    DwellTimer(IN:=TRUE, PT:= T#10S);
	IF (DwellTimer.Q) THEN
		ErrorReturnState := ePistonInsertStaState.eRetractPalletHoldDownAndBarrel;		
		ResetDwellTimer();
		ResetStateTimer();
		NextState := ePistonInsertStaState.eError;		
	END_IF 
  

ePistonInsertStaState.eDepart:
	StateTimer(IN:=TRUE, PT:= T#20MS);
	IF (StateTimer.Q) THEN
		Stations.fbRoutePlanner.M_NotifyVehStaCmpl(StationIndex:= MM_CONST.PISTON_STA, VehicleID := VUT);
		xTrigger := FALSE;	
		StateTimer(IN:=FALSE);
		IF (NOT Stations.fbCycleControl.StopRequested) THEN			
			NextState := ePistonInsertStaState.eInit;
		ELSE 
			NextState := ePistonInsertStaState.eStopActive;
		END_IF
	END_IF

ePistonInsertStaState.eStopActive:
IF (NOT Stations.fbCycleControl.StopRequested) THEN			
	NextState := ePistonInsertStaState.eInit;
END_IF	
Status.PistonStatusMsg:= 'Piston Sta Cycle Stop, Hit Start'; 
	
ePistonInsertStaState.eError:
	Status.StationStauts[MM_CONST.PISTON_STA_HMI_STATE] := OverallStationStatus.eError;
	IF (GVL_IO.MC_XStartPB) THEN
		NextState := ErrorReturnState;
		ErrorReturnState := ePistonInsertStaState.eUnknown;
	END_IF

END_CASE

IF (State <> NextState) THEN
	bFirst := TRUE;
	StateTimer(IN:=FALSE);
ELSE
	bFirst := FALSE;
END_IF

State := NextState;
AssignStationStatusForHMI();

ACTION Act_EngagePalletHoldDown:
GVL_IO.PI_YPalletHoldDownExtend:= TRUE;
GVL_IO.PI_YPalletHoldDownRetract := FALSE;
END_ACTION

ACTION Act_ExtendBarrelBackup:
GVL_IO.PI_YBarrelBackupExtend := TRUE;
GVL_IO.PI_YBarrelBackupRetract := FALSE;
END_ACTION

ACTION Act_FreePalletHoldDown:
GVL_IO.PI_YPalletHoldDownExtend:= FALSE;
GVL_IO.PI_YPalletHoldDownRetract := TRUE;
END_ACTION

ACTION Act_RetractBarrelBackup:
GVL_IO.PI_YBarrelBackupExtend := FALSE;
GVL_IO.PI_YBarrelBackupRetract := TRUE;
END_ACTION

ACTION Act_SendEscapementToBowl:
GVL_IO.PI_YEscapementToBowl := TRUE;
GVL_IO.PI_YEscapementToWork := FALSE;
END_ACTION

ACTION Act_SendEscapementtoWork:
GVL_IO.PI_YEscapementToBowl := FALSE;
GVL_IO.PI_YEscapementToWork := TRUE;
END_ACTION

METHOD PUBLIC AssignStationStatusForHMI : BOOL
VAR_INPUT
END_VAR
Status.StationsState[MM_CONST.PISTON_STA_HMI_STATE] := State;
IF (NOT LotsData.Lot.PistonInsertEnabled AND NOT (State = ePistonInsertStaState.eUnknown) AND NOT (State = ePistonInsertStaState.eError)) THEN
	Status.StationStauts[MM_CONST.PISTON_STA_HMI_STATE] := OverallStationStatus.eDisabled;
ELSE 
	CASE State OF 
	ePistonInsertStaState.eUnknown,ePistonInsertStaState.eError: 
		Status.StationStauts[MM_CONST.PISTON_STA_HMI_STATE] := OverallStationStatus.eError;
	 
    
    ePistonInsertStaState.eSMCMtrReset,ePistonInsertStaState.eSMCMtrCheckEnabled,ePistonInsertStaState.eSMCMtrSendHome,
    ePistonInsertStaState.eSMCMtrHomed,ePistonInsertStaState.eInit, ePistonInsertStaState.eHoming,
	ePistonInsertStaState.eMoveEscapemttoBowl,
	ePistonInsertStaState.eEscapmentAtBowl,
	ePistonInsertStaState.eMoveEscapmentToWork,
	ePistonInsertStaState.eEscapementAtWork:
    	Status.StationStauts[MM_CONST.PISTON_STA_HMI_STATE] := OverallStationStatus.eHoming;	
	
	ePistonInsertStaState.eWaitForPartAtBowl:
		Status.StationStauts[MM_CONST.PISTON_STA_HMI_STATE] := OverallStationStatus.eWarning;
	
	ePistonInsertStaState.eReady:
		Status.StationStauts[MM_CONST.PISTON_STA_HMI_STATE] := OverallStationStatus.eWaitingForParts;
	
	ePistonInsertStaState.ePalletHoldDownEngaged,
	ePistonInsertStaState.eFirePistonUp,
	ePistonInsertStaState.eSendBarrelBackupEngage,
	ePistonInsertStaState.eWaitForPistonStartMovUp,
	ePistonInsertStaState.eWaitForBarrelBackupEngaged,
	ePistonInsertStaState.eWaitForPistonMovDoneUp,
	ePistonInsertStaState.eFirePistonDown,
	ePistonInsertStaState.eRetractPalletHoldDownAndBackup,
	ePistonInsertStaState.eWaitForPistonStartMovDwn,
	ePistonInsertStaState.eRetractPalletHoldDownAndBarrel,
	ePistonInsertStaState.eWaitForPalletHoldDownAndBackupRetracted,
	ePistonInsertStaState.eWaitForPistonMovDoneDown :
		Status.StationStauts[MM_CONST.PISTON_STA_HMI_STATE] := OverallStationStatus.eWaitingForParts; 
	
    ePistonInsertStaState.eStopActive:
	    Status.StationStauts[MM_CONST.PISTON_STA_HMI_STATE] := OverallStationStatus.eCycleStop;
	 
	ELSE ;
	
	END_CASE
END_IF
END_METHOD

METHOD PUBLIC ClearVehicleTrigger : BOOL
VAR_INPUT
END_VAR
xTrigger := FALSE;
END_METHOD

METHOD PUBLIC IsBarrelBackupExtended : BOOL
VAR_INPUT
END_VAR
IsBarrelBackUpExtended := TRUE;  // IMBAD 2 Has No Barrel Backup
(*
IsBarrelBackUpExtended := GVL_IO.PI_XBarrelHoldDownExtended AND NOT GVL_IO.PI_XBarrelHoldDownHome;
IF (NOT IsBarrelBackUpExtended) THEN
	Status.PistonStatusMsg := 'Piston: Check Barrel Backup Sensors';
END_IF
*)
END_METHOD

METHOD PUBLIC IsBarrelBackUpRetracted : BOOL
VAR_INPUT
END_VAR
IsBarrelBackUpRetracted := TRUE;  // IMBAD 2 has no Barrel Backup
(* 
IsBarrelBackUpRetracted := NOT GVL_IO.PI_XBarrelHoldDownExtended AND GVL_IO.PI_XBarrelHoldDownHome;
IF (NOT IsBarrelBackUpRetracted) THEN
	Status.PistonStatusMsg := 'Piston: Check Barrel Backup Sensors';
END_IF
*)
END_METHOD

METHOD PUBLIC IsEscapementAtBowl : BOOL
VAR_INPUT
END_VAR
IsEscapementAtBowl := (GVL_IO.PI_XEscapementAtBowl);// AND NOT GVL_IO.PI_XEscapementAtInsertLoc);
IF (NOT IsEscapementAtBowl) THEN
	Status.PistonStatusMsg := 'Piston: Check Escapment Sensors';
END_IF
END_METHOD

METHOD PUBLIC IsEscapementAtWork : BOOL
VAR_INPUT
END_VAR
IsEscapementAtWork := ((*NOT GVL_IO.PI_XEscapementAtBowl AND *)GVL_IO.PI_XEscapementAtInsertLoc);
IF (NOT IsEscapementAtWork) THEN
	Status.PistonStatusMsg := 'Piston: Check Escapment Sensors';
END_IF
END_METHOD

METHOD PUBLIC IsFaulted : BOOL
VAR_INPUT
END_VAR
IsFaulted := (State = ePistonInsertStaState.eUnknown OR State = ePistonInsertStaState.eError);
END_METHOD

METHOD PUBLIC IsPalletHoldDownEngaged : BOOL
VAR_INPUT
END_VAR
IsPalletHoldDownEngaged := (NOT GVL_IO.PI_XPalletHoldDownHome (*AND GVL_IO.PI_XPalletHoldDownExtended*));
IF (NOT IsPalletHoldDownEngaged) THEN
	Status.PistonStatusMsg := 'Piston: Check Pallet Hold Down'; 
END_IF
END_METHOD

METHOD PUBLIC IsPalletHoldDownFree : BOOL
VAR_INPUT
END_VAR
IsPalletHoldDownFree := (GVL_IO.PI_XPalletHoldDownHome AND NOT GVL_IO.PI_XPalletHoldDownExtended);
IF (NOT IsPalletHoldDownFree) THEN
	Status.PistonStatusMsg := 'Piston: Check Pallet Hold Down'; 
END_IF
END_METHOD

METHOD PUBLIC LEY_MasterReset : BOOL
VAR_INPUT
END_VAR
GVL_IO.PI_YMtrReset := TRUE;
GVL_IO.PI_YMtrSetEnable:= TRUE;
GVL_IO.PI_YMtrDriveStepTrigger := FALSE;
GVL_IO.PI_YMtrHoldMove := FALSE;
GVL_IO.PI_YMtrGoHome := FALSE;
GVL_IO.PI_YMtrJogNeg := FALSE;
GVL_IO.PI_YMtrJogPos := FALSE;
GVL_IO.PI_YMtrSwitchJogInch := FALSE;
GVL_IO.PI_YMtrStepSelectIN0:= FALSE;
GVL_IO.PI_YMtrStepSelectIN1:= FALSE;
GVL_IO.PI_YMtrStepSelectIN2:= FALSE;
GVL_IO.PI_YMtrStepSelectIN3:= FALSE;
GVL_IO.PI_YMtrStepSelectIN4:= FALSE;
GVL_IO.PI_YMtrStepSelectIN5:= FALSE;
END_METHOD

PROPERTY PUBLIC Ready : BOOL
GET
IF (LotsData.Lot.PistonInsertEnabled) THEN
	Ready := (State = ePistonInsertStaState.eReady);
ELSE
    Ready := (State = ePistonInsertStaState.eDisabledReady);
END_IF
END_GET
END_PROPERTY

ACTION ResetDwellTimer:
DwellTimer(IN:=FALSE);
END_ACTION

METHOD PUBLIC ResetState : BOOL
VAR_INPUT
END_VAR
	State := ePistonInsertStaState.eUnknown;
	NextState := ePistonInsertStaState.eUnknown;
END_METHOD

ACTION ResetStateTimer:
StateTimer(IN:=FALSE);
END_ACTION

PROPERTY PUBLIC Trigger : BOOL
SET
xTrigger := Trigger;
END_SET
END_PROPERTY

METHOD PUBLIC UpdatePartData : BOOL
VAR_INPUT
END_VAR
PartsData.Status[VUT].OverallStatus := ePartStatus.ePistonInserted;
PartsData.Status[VUT].PistonStroke := GVL_IO.PI_XMtrCurrPos;
PartsData.Status[VUT].PistonPass := TRUE;
PartsData.Status[VUT].PistonInsertTime := SYSTEMTIME_TO_STRING(Logging.fbCurrTime.systemTime);
END_METHOD

PROPERTY PUBLIC VehicleUnderTest : BYTE
GET
VehicleUnderTest := VUT;
END_GET
SET
VUT := VehicleUnderTest;
END_SET
END_PROPERTY

END_FUNCTION_BLOCK

// ---- POUs/IB_StopRobotClearStation.TcPOU
FUNCTION_BLOCK PUBLIC IB_StopRobotClearStation
VAR_INPUT
END_VAR
VAR_OUTPUT
END_VAR
VAR
	xTrigger :BOOL := FALSE; // triggers processing
	State : eIB_StopRobotClearStaState := eIB_StopRobotClearStaState.eUnknown;
	NextState : eIB_StopRobotClearStaState := eIB_StopRobotClearStaState.eUnknown;
	bFirst : BOOL := TRUE;
	VUT : BYTE; //VehicleID Under Station
	DwellTimer : TON;
END_VAR

CASE State OF
eIB_StopRobotClearStaState.eUnknown:
	NextState := eIB_StopRobotClearStaState.eReady;
	
eIB_StopRobotClearStaState.eInit:

eIB_StopRobotClearStaState.eHoming:

eIB_StopRobotClearStaState.eReady:
	IF (xTrigger) THEN
		NextState := eIB_StopRobotClearStaState.eProcessing;		
		DwellTimer(IN:=FALSE);
	END_IF

eIB_StopRobotClearStaState.eDwell:	

eIB_StopRobotClearStaState.eProcessing:
	IF(Stations.fbLoad1Sta.HoldVehicle_IBStop = FALSE) THEN
		NextState := eIB_StopRobotClearStaState.eDepart;
	END_IF

eIB_StopRobotClearStaState.eDepart:
		Stations.fbRoutePlanner.M_NotifyVehStaCmpl(StationIndex:= MM_CONST.IB_STOP_ROBOT_CLEAR_STA, VehicleID := VUT);
		xTrigger := FALSE;
		IF (Stations.fbCycleControl.StopRequested) THEN
			NextState := eIB_StopRobotClearStaState.eStopActive;
		ELSE
			NextState := eIB_StopRobotClearStaState.eReady;		
		END_IF
		
eIB_StopRobotClearStaState.eStopActive:
	IF (NOT Stations.fbCycleControl.StopRequested) THEN
		NextState := eIB_StopRobotClearStaState.eReady;	
	END_IF
		
eIB_StopRobotClearStaState.eError:
END_CASE

IF (State <> NextState) THEN
	bFirst := TRUE;
ELSE
	bFirst := FALSE;
END_IF

State := NextState;
//Status.StationsState[MM_CONST.IB_STOP_ROBOT_CLEAR_STA_HMI_STATE] := State;
//AssignStationStatusForHMI();

METHOD PUBLIC ClearVehicleTrigger : BOOL
VAR_INPUT
END_VAR
xTrigger := FALSE;
State  := eIB_StopRobotClearStaState.eUnknown;
NextState  := eIB_StopRobotClearStaState.eUnknown;
bFirst  := TRUE;
END_METHOD

PROPERTY PUBLIC Trigger : BOOL
SET
xTrigger := Trigger;
END_SET
END_PROPERTY

PROPERTY PUBLIC VehicleUnderTest : BYTE
GET
VehicleUnderTest := VUT;
END_GET
SET
VUT := VehicleUnderTest;
END_SET
END_PROPERTY

END_FUNCTION_BLOCK

// ---- POUs/CapInsertStation.TcPOU
FUNCTION_BLOCK PUBLIC CapInsertStation
VAR_INPUT
END_VAR
VAR_OUTPUT
END_VAR
VAR
	xTrigger :BOOL := FALSE; // triggers processing
	State : eCapInsertStaState := eCapInsertStaState.eUnknown;
	NextState : eCapInsertStaState := eCapInsertStaState.eUnknown;
	ErrorReturnState :  eCapInsertStaState := eCapInsertStaState.eUnknown;
	bFirst : BOOL := TRUE;
	VUT : BYTE; //VehicleID Under Station
	DwellTimer : TON;		
	StateTimer : TON;
	PartPresentTimer : TON;
	CapInstallRetries : BYTE :=0;
	CapPickUpRetries : BYTE := 0;
	CapTorqueTime : TIME := T#250MS;
END_VAR

/// Cap station can be either Disabled or Enabled
// If Disabled, then we need to be in a state such that it is disabled but will not cause any obstacles. 
// Either in Disabled - Ready or Enabled- Ready, provide a way to account for Station enable change

IF (GVL_IO.MachineEStopped) THEN 
	State := eCapInsertStaState.eUnknown;
	NextState := eCapInsertStaState.eUnknown;	
END_IF

CASE State OF

eCapInsertStaState.eUnknown:
	   IF (GVL_IO.MC_XStartPB AND GVL_IO.MC_XAirPressureOK AND GVL_IO.MC_NotEStopped) THEN // wait for start button when powered up or PLC program restarted
		 ResetDwellTimer();	
         NextState := eCapInsertStaState.eHoming;	              
	   END_IF
	ACT_RetractSlide();
	ACT_RetractPalletHoldDown();
	Status.CapStatusMsg:= 'CapSta Unknown,Check Air/E-STOP THEN Hit Start';

eCapInsertStaState.eHoming:
    Status.StationStauts[MM_CONST.CAP_STA_HMI_STATE] := OverallStationStatus.eHoming;
	Status.CapStatusMsg:= 'Cap Station Homing';
	
	ACT_RetractSlide();
	ACT_RetractPalletHoldDown();
	DwellTimer(IN:=TRUE, PT:= T#10S);	
	IF (IsPalletHoldDownRetracted() AND IsSlideRetracted()) THEN
		ResetDwellTimer();	
		IF (NOT LotsData.Lot.CapInsertEnabled) THEN
			NextState :=  eCapInsertStaState.eDisabledReady;			
        ELSE 
            NextState :=  eCapInsertStaState.eWaitForVehicleTrigger;
		END_IF
	END_IF
    IF (DwellTimer.Q) THEN
		ResetDwellTimer();
		NextState := eCapInsertStaState.eError;
		ErrorReturnState := eCapInsertStaState.eHoming;		
	END_IF
	
	

eCapInsertStaState.eDisabledReady:
	ACT_RetractSlide();
	ACT_RetractPalletHoldDown();
	IF (LotsData.Lot.CapInsertEnabled) THEN 
		NextState := eCapInsertStaState.eUnknown; // force the operator to hit the start button if station is enabled.
	END_IF
	IF (xTrigger) THEN // vehicles that have been previously commanded to come here before station was disabled 
		NextState := eCapInsertStaState.eDepart;
	END_IF
	Status.StationStauts[MM_CONST.CAP_STA_HMI_STATE] := OverallStationStatus.eDisabled;
	Status.CapStatusMsg:= 'Cap Station Disabled and Clear for pallets to move';
	
	
eCapInsertStaState.eWaitForVehicleTrigger:
  
	IF (xTrigger) THEN //XTrigger is signaled when part arrives under the station
		NextState := eCapInsertStaState.ePalletHoldDownGoingDown;	
	    PartsData.Status[VUT].OverallStatus := ePartStatus.eReject; 		
		ResetDwellTimer();
	END_IF
	
	Status.StationStauts[MM_CONST.CAP_STA_HMI_STATE] := OverallStationStatus.eWaitingForParts;
	Status.CapStatusMsg:= 'Cap Station Waiting For Parts';

eCapInsertStaState.ePalletHoldDownGoingDown:
	ACT_EngagePalletHoldDown();
	IF (IsPalletHoldDownExtended()) THEN
		   NextState := eCapInsertStaState.ePalletHoldDownExtended;		 
           ResetDwellTimer();  
	   END_IF
	DwellTimer(IN:=TRUE, PT:= T#10S); // give a message out every 10 seconds
	IF (DwellTimer.Q) THEN
		ResetDwellTimer();
		NextState := eCapInsertStaState.eError;
		ErrorReturnState := eCapInsertStaState.ePalletHoldDownGoingDown;			
	END_IF
	
	Status.StationStauts[MM_CONST.CAP_STA_HMI_STATE] := OverallStationStatus.eRunning;
	Status.CapStatusMsg:= 'Cap Cycle In Progress';
	
eCapInsertStaState.ePalletHoldDownExtended:
   DwellTimer(IN:=TRUE, PT:= T#250MS);
   IF (DwellTimer.Q) THEN 
	   ResetDwellTimer();
       NextState := eCapInsertStaState.eCapSlideGoingDown;
   END_IF

eCapInsertStaState.eCapSlideGoingDown:
   ACT_ExtendSlide();
   IF (NOT IsSlideRetracted()) THEN 
	   NextState := eCapInsertStaState.eCapSlideExtended;
	   ResetDwellTimer();
   END_IF
   DwellTimer(IN:=TRUE, PT:= T#5S); // give a message out every 10 seconds
	IF (DwellTimer.Q) THEN
		ResetDwellTimer();
		Act_RetractSlide();  // Not wanting to spin the cap station if case of time out
		NextState := eCapInsertStaState.eError;
		ErrorReturnState := eCapInsertStaState.eCapSlideGoingDown;			
	END_IF

eCapInsertStaState.eCapSlideExtended:
   DwellTimer(IN:=TRUE, PT:= CapTorqueTime);
   IF (DwellTimer.Q OR IsSlideExtended()) THEN 
	   ResetDwellTimer();
	   UpdatePartData();	   
       NextState := eCapInsertStaState.eCapSlideGoingUp;
   END_IF

 eCapInsertStaState.eCapSlideGoingUp:
   ACT_RetractSlide();
   ResetDwellTimer();
   NextState := eCapInsertStaState.eCapSlideUp;
   
eCapInsertStaState.eCapSlideUp:
    IF (IsSlideRetracted()) THEN
	   ResetDwellTimer();
	   NextState := eCapInsertStaState.ePalletHoldDownGoingUp;
   END_IF
   
    DwellTimer(IN:=TRUE, PT:= T#10S); 
	IF (DwellTimer.Q) THEN
		ResetDwellTimer();
		NextState := eCapInsertStaState.eError;
		ErrorReturnState := eCapInsertStaState.eCapSlideGoingUp;			
	END_IF
   
eCapInsertStaState.ePalletHoldDownGoingUp:
	ACT_RetractPalletHoldDown();
	ResetDwellTimer();
	NextState := eCapInsertStaState.ePalletHoldDownUp;

eCapInsertStaState.ePalletHoldDownUp:
  
   IF (IsPalletHoldDownRetracted()) THEN
	   ResetDwellTimer();
	   NextState := eCapInsertStaState.eDepart;
   END_IF 
    DwellTimer(IN:=TRUE, PT:= T#10S); // give a message out every 10 seconds
	IF (DwellTimer.Q) THEN
		ResetDwellTimer();
		NextState := eCapInsertStaState.eError;
		ErrorReturnState := eCapInsertStaState.ePalletHoldDownGoingUp;			
	END_IF


eCapInsertStaState.eDepart:
	Stations.fbRoutePlanner.M_NotifyVehStaCmpl(StationIndex:= MM_CONST.CAP_STA, VehicleID := VUT);
	xTrigger := FALSE; // Now that we have sent a vehicle out, we should not work on it anymore 
    IF (Stations.fbCycleControl.StopRequested) THEN		
		NextState := eCapInsertStaState.eStopActive;
	ELSE
		NextState := eCapInsertStaState.eHoming;
	END_IF

eCapInsertStaState.eStopActive:
IF (NOT Stations.fbCycleControl.StopRequested) THEN		
		NextState := eCapInsertStaState.eHoming;
END_IF	
    Status.StationStauts[MM_CONST.CAP_STA_HMI_STATE] := OverallStationStatus.eCycleStop;	
    Status.CapStatusMsg:= 'Cap Stop Active, Press Start to Run';
	
eCapInsertStaState.eError:
	Status.StationStauts[MM_CONST.CAP_STA_HMI_STATE] := OverallStationStatus.eError;
	IF (GVL_IO.MC_XStartPB) THEN
		NextState := ErrorReturnState;
		ErrorReturnState := eCapInsertStaState.eUnknown;
	END_IF
	
END_CASE

IF (State <> NextState) THEN
	bFirst := TRUE;
	StateTimer(IN:=FALSE);
ELSE
	bFirst := FALSE;
END_IF

State := NextState;

ACTION ACT_EngagePalletHoldDown:
GVL_IO.CP_YPalletHoldDownExtend := TRUE;
GVL_IO.CP_YPalletHoldDownRetract := FALSE;
END_ACTION

ACTION ACT_ExtendSlide:
GVL_IO.CP_YCapSlideExtend := TRUE;
GVL_IO.CP_YCapSlideRetract := FALSE;
END_ACTION

ACTION ACT_RetractPalletHoldDown:
GVL_IO.CP_YPalletHoldDownExtend := FALSE;
GVL_IO.CP_YPalletHoldDownRetract := TRUE;
END_ACTION

ACTION ACT_RetractSlide:
GVL_IO.CP_YCapSlideExtend := FALSE;
GVL_IO.CP_YCapSlideRetract := TRUE;
END_ACTION

METHOD PUBLIC ClearVehicleTrigger : BOOL
VAR_INPUT
END_VAR
xTrigger := FALSE;
END_METHOD

METHOD PUBLIC IsFaulted : BOOL
VAR_INPUT
END_VAR
IF (LotsData.Lot.CapInsertEnabled) THEN 
	IsFaulted := (State = eCapInsertStaState.eUnknown OR State = eCapInsertStaState.eError);
ELSE 
	IsFaulted := FALSE;
END_IF
END_METHOD

METHOD PUBLIC IsPalletHoldDownExtended : BOOL
VAR_INPUT
END_VAR
IsPalletHoldDownExtended := (GVL_IO.CP_XPalletHoldDownExtended AND NOT GVL_IO.CP_XPalletHoldDownHome);
IF (NOT IsPalletHoldDownExtended) THEN 
	Status.CapStatusMsg := 'Cap Station: Check Pallet HoldDown Sensors'; 
END_IF
END_METHOD

METHOD PUBLIC IsPalletHoldDownRetracted : BOOL
VAR_INPUT
END_VAR
IsPalletHoldDownRetracted := (NOT GVL_IO.CP_XPalletHoldDownExtended AND GVL_IO.CP_XPalletHoldDownHome);
IF (NOT IsPalletHoldDownRetracted) THEN 
	Status.CapStatusMsg := 'Cap Station: Check Pallet HoldDown Sensors'; 
END_IF
END_METHOD

METHOD IsSlideExtended : BOOL
VAR_INPUT
END_VAR
IsSlideExtended := (GVL_IO.CP_XCapSlideExtended AND NOT GVL_IO.CP_XCapSlideRetracted);
IF (NOT IsSlideExtended) THEN 
	Status.CapStatusMsg := 'Cap Station: Check Slide Sensors'; 
END_IF
END_METHOD

METHOD PUBLIC IsSlideRetracted : BOOL
VAR_INPUT
END_VAR
//IsSlideRetracted := TRUE; //turnkey slide removed

IsSlideRetracted := (NOT GVL_IO.CP_XCapSlideExtended AND GVL_IO.CP_XCapSlideRetracted);
IF (NOT IsSlideRetracted) THEN 
	Status.CapStatusMsg := 'Cap Station: Check Slide Sensors'; 
END_IF
END_METHOD

PROPERTY PUBLIC Ready : BOOL
GET
IF (LotsData.Lot.CapInsertEnabled) THEN
 Ready := (State = eCapInsertStaState.eWaitForVehicleTrigger);
ELSE
	Ready := (State = eCapInsertStaState.eDisabledReady);	//we removed the physical cap station on 10/17 
END_IF
END_GET
END_PROPERTY

ACTION ResetDwellTimer:
DwellTimer(IN:=FALSE);
END_ACTION

METHOD PUBLIC ResetState : BOOL
VAR_INPUT
END_VAR
	State := eCapInsertStaState.eUnknown;
	NextState := eCapInsertStaState.eUnknown;
	ErrorReturnState := eCapInsertStaState.eUnknown;
END_METHOD

PROPERTY PUBLIC Trigger : BOOL
SET
xTrigger := Trigger;
END_SET
END_PROPERTY

METHOD PUBLIC UpdatePartData : BOOL
VAR_INPUT
END_VAR
IF ( NOT IsSlideExtended()) THEN
	PartsData.Status[VUT].OverallStatus := ePartStatus.eCapInserted;
	PartsData.Status[VUT].CapPass := TRUE;
	PartsData.Status[VUT].CapInsertTime := SYSTEMTIME_TO_STRING(Logging.fbCurrTime.systemTime);	
ELSE // there is no cap
	PartsData.Status[VUT].OverallStatus := ePartStatus.eReject;
	PartsData.Status[VUT].CapPass := FALSE;
	PartsData.Status[VUT].CapInsertTime := SYSTEMTIME_TO_STRING(Logging.fbCurrTime.systemTime);
END_IF
END_METHOD

PROPERTY PUBLIC VehicleUnderTest : BYTE
GET
VehicleUnderTest := VUT;
END_GET
SET
VUT := VehicleUnderTest;
END_SET
END_PROPERTY

END_FUNCTION_BLOCK

// ---- POUs/GoodUnloadStation.TcPOU
FUNCTION_BLOCK PUBLIC GoodUnloadStation
VAR_INPUT
END_VAR
VAR_OUTPUT
END_VAR
VAR
	xTrigger :BOOL := FALSE; // triggers processing
	State : eGoodULStaState := eGoodULStaState.eUnknown;
	NextState : eGoodULStaState := eGoodULStaState.eUnknown;	
	ErrorReturnState : eGoodULStaState := eGoodULStaState.eUnknown;	
	bFirst : BOOL := TRUE;
	VUT : BYTE; //VehicleID Under Station
	DwellTimer : TON;
	StateTimer : TON;
	eDwell: INT;
	eDepart: INT;
	CurrPPLoc : BYTE;
	GripperOpenTimer :TIME := T#200MS;
	//StopAfter
	DropLocation : BYTE;
	GoodFullCount : UINT := 0;
	PremiumFullCount : UINT := 0;
	
END_VAR

IF (GVL_IO.MachineEStopped) THEN 
	State := eGoodULStaState.eUnknown;
	NextState := eGoodULStaState.eUnknown;	
	Status.GoodULStatusMsg:= 'Unload: Unknown State, Check E-STOP, Check Air, Hit Start';
END_IF

GetPPLocation(Location=>CurrPPLoc); // Get where PP Location is from the Bits. 

IF (NOT LotsData.Lot.AutoBaggerEnabled) THEN
	Config.PremiumCount1 := 0;
	Config.PremiumCount2 := 0;
	Config.GoodCount1 := 0;
	Config.GoodCount2 := 0;
	GoodFullCount := 0;
    PremiumFullCount := 0;
END_IF


CASE State OF
	
eGoodULStaState.eUnknown:
	IF (GVL_IO.MC_XStartPB AND GVL_IO.MC_XAirPressureOK AND GVL_IO.MC_NotEStopped) THEN // wait for start button when powered up or PLC program restarted
			NextState := eGoodULStaState.eInit;	   
	END_IF

eGoodULStaState.eInit:
    Act_OpenGrippers();
	Act_FreePalletHold();
	Act_FreePalletRelease();
    Act_MoveRotatorCenter();
	Act_ResetPPIO();	
	
	StateTimer(IN:=TRUE,PT:= T#100MS);
	IF (StateTimer.Q) THEN
		NextState := eGoodULStaState.eHoming;
		ResetStateTimer();
	END_IF	

eGoodULStaState.eHoming:
  
	IF (IsGripperOpen() AND IsPalletReleaseFree() AND IsRotatorCenter() AND IsPalletHoldDownFree()) THEN
	  NextState := eGoodULStaState.eHPReset;
	  ResetDwellTimer();
 	END_IF	
	
   DwellTimer(IN:=TRUE, PT:= T#10S);
   IF (DwellTimer.Q) THEN
		ErrorReturnState := eGoodULStaState.eInit;		
		ResetDwellTimer();
		ResetStateTimer();
        NextState := eGoodULStaState.eError;		
	END_IF
	

eGoodULStaState.eHPReset:
	IF (GVL_IO.UL_XPP_Alarm) THEN
		DwellTimer(IN:= TRUE, PT := T#2S);	
	END_IF
	IF (DwellTimer.Q) THEN
		ResetDwellTimer();
		GVL_IO.UL_YPP_ResetAlarm := NOT GVL_IO.UL_YPP_ResetAlarm; // toggle the reset request every four seconds 
	END_IF
	IF (NOT GVL_IO.UL_XPP_Alarm) THEN
		GVL_IO.UL_YPP_Enable:= TRUE;
		GVL_IO.UL_YPP_ResetAlarm := FALSE;
		ResetDwellTimer();
		NextState := eGoodULStaState.eHPCheckEnabled;	
	END_IF
	// Time out condition... hang here until Pick Place Alarm is reset... 
	DwellTimer(IN:=TRUE, PT:= T#10S);
   IF (DwellTimer.Q) THEN
		ErrorReturnState := eGoodULStaState.eHPReset;		
		ResetDwellTimer();
		ResetStateTimer();
		Status.GoodULStatusMsg:= 'Pick&Place unable to Reset';
        NextState := eGoodULStaState.eError;		
	END_IF

eGoodULStaState.eHPCheckEnabled:
	IF (GVL_IO.UL_XPP_DriveEnabled AND NOT GVL_IO.UL_XPP_Alarm) THEN
		ResetDwellTimer();
        IF (GVL_IO.UL_XPP_ReferenceOK) THEN
			NextState := eGoodULStaState.eHPHomed;			
			GVL_IO.UL_YPP_StartHoming := FALSE;
		ELSE			
			NextState := eGoodULStaState.eHPSendHome;
		END_IF
	END_IF
	
	// Time out condition... hang here until Pick Place Alarm is reset... 
   DwellTimer(IN:=TRUE, PT:= T#10S);
   IF (DwellTimer.Q) THEN
		ErrorReturnState := eGoodULStaState.eHPReset;		
		ResetDwellTimer();
		ResetStateTimer();
		Status.GoodULStatusMsg:= 'Pick&Place unable to Enable';
        NextState := eGoodULStaState.eError;		
	END_IF

eGoodULStaState.eHPSendHome:
	GVL_IO.UL_YPP_Stop := FALSE;
	IF (NOT GVL_IO.UL_XPP_StopActive AND GVL_IO.UL_XPP_ReadyToStart AND GVL_IO.UL_XPP_DriveEnabled AND NOT GVL_IO.UL_XPP_Alarm) THEN
		GVL_IO.UL_YPP_StartHoming := TRUE;
	END_IF
	
   IF (GVL_IO.UL_XPP_ReferenceOK) THEN
	   NextState := eGoodULStaState.eHPHomed;
	   ResetDwellTimer();
   END_IF
   
   DwellTimer(IN:=TRUE, PT:= T#2M);
   IF (DwellTimer.Q) THEN
		ErrorReturnState := eGoodULStaState.eInit;		
		ResetDwellTimer();
		ResetStateTimer();
		GVL_IO.UL_YPP_StartHoming := FALSE;
		Status.GoodULStatusMsg:= 'Pick&Place unable to Home';
        NextState := eGoodULStaState.eError;		
	END_IF
 

eGoodULStaState.eHPHomed:
	GVL_IO.UL_YPP_Stop := FALSE;
	GVL_IO.UL_YPP_Enable := TRUE;
	GVL_IO.UL_YPP_StartHoming := FALSE;
	IF (GVL_IO.UL_XPP_ReadyToStart) THEN
		NextState := eGoodULStaState.eHPSendToInitLoc;
		ResetDwellTimer();
		ResetStateTimer();
	END_IF
	
    DwellTimer(IN:=TRUE, PT:= T#2M);
   IF (DwellTimer.Q) THEN
		ErrorReturnState := eGoodULStaState.eHPReset;		
		ResetDwellTimer();
		ResetStateTimer();
		GVL_IO.UL_YPP_StartHoming := FALSE;
		Status.GoodULStatusMsg:= 'Pick&Place unable to Ready To Start';
        NextState := eGoodULStaState.eError;		
	END_IF

eGoodULStaState.eHPSendToInitLoc:
   // we have to set Seq 1 as InitLoc ( Up at Pick Location). Also, Input bits will corresponding to the sequence 
   SetPPSequence(SequenceNumb := 1);
   DwellTimer(IN:= TRUE, PT:= T#30MS);
   IF (DwellTimer.Q) THEN
	   GVL_IO.UL_YPP_StartSeq := TRUE;
	   ResetDwellTimer();
   END_IF
   StateTimer(IN:= GVL_IO.UL_YPP_StartSeq, PT:= T#30MS);
   IF (StateTimer.Q) THEN
	   NextState := eGoodULStaState.eHPAtInitLoc;
	   ResetStateTimer();
	   ResetDwellTimer();
   END_IF
 
eGoodULStaState.eHPAtInitLoc:
	IF (CurrPPLoc = 1) THEN
		NextState:= eGoodULStaState.eHPReady;
		GVL_IO.UL_YPP_StartSeq := FALSE;
		ResetDwellTimer();
		ResetStateTimer();
	END_IF
   DwellTimer(IN:=TRUE, PT:= T#10S);
   IF (DwellTimer.Q) THEN
		ErrorReturnState := eGoodULStaState.eHPSendToInitLoc;		
		ResetDwellTimer();
		ResetStateTimer();
		GVL_IO.UL_YPP_StartSeq := FALSE;
		Status.GoodULStatusMsg:= 'Pick&Place unable to Go To Init Loc';
        NextState := eGoodULStaState.eError;		
	END_IF

eGoodULStaState.eHPReady:
    Status.GoodULStatusMsg:= 'Unload Ready';
    Act_OpenGrippers();
	Act_FreePalletHold();
    Act_FreePalletRelease();
    Act_MoveRotatorCenter();	
	//PP fieldbus commands
	SetPPSequence(SequenceNumb := 1);
	Act_EnablePP();
	GVL_IO.UL_YPP_StartSeq := FALSE;
	
	 IF (IsGripperOpen() AND IsPalletReleaseFree() AND IsRotatorCenter() AND IsPalletHoldDownFree() AND GVL_IO.UL_XPP_ReadyToStart ) THEN
	  	 ResetDwellTimer();
         IF (LotsData.Lot.GoodUnloadEnabled) THEN
			 NextState:= eGoodULStaState.eWaitForVehicleTrigger;			 
		 ELSE 
			 NextState := eGoodULStaState.eDisabledReady;
		 END_IF    
    END_IF	
	
	DwellTimer(IN:=TRUE, PT:= T#10S);
   IF (DwellTimer.Q) THEN
		ErrorReturnState := eGoodULStaState.eHPReady;		
		ResetDwellTimer();
		ResetStateTimer();				
        NextState := eGoodULStaState.eError;		
	END_IF
	
	

eGoodULStaState.eDisabledReady:
	
	IF (LotsData.Lot.GoodUnloadEnabled) THEN
		NextState := eGoodULStaState.eUnknown;
	END_IF
	IF (xTrigger) THEN
		Stations.fbRoutePlanner.M_NotifyVehStaCmpl(StationIndex:= MM_CONST.GOOD_UNLOAD_STA, VehicleID := VUT);
		xTrigger := FALSE;
		NextState := eGoodULStaState.eDepartVehicle;
	END_IF

eGoodULStaState.eWaitForVehicleTrigger:

	IF (xTrigger) THEN //XTrigger is signaled when part arrives under the station
		DwellTimer(IN:=TRUE, PT:= T#100MS);
        IF (DwellTimer.Q) THEN 
			NextState := eGoodULStaState.eDetermineDropLocation;
			ResetDwellTimer();
        END_IF								
	END_IF
	
	IF (NOT LotsData.Lot.GoodUnloadEnabled) THEN
		NextState := eGoodULStaState.eDisabledReady;
	END_IF
	
	Status.GoodULStatusMsg:= 'Unload Ready: Waiting For Vehicle';
		 
eGoodULStaState.eDetermineDropLocation: //Determine drop locations.  Premiums can go in good if Premium is full.  

	IF (PartsData.Status[VUT].Premium) THEN
		IF (NOT LotsData.Lot.AutoBaggerEnabled) THEN
			DropLocation := 1;
			NextState := eGoodULStaState.eDwell;
		ELSIF ((Config.PremiumCount1 < LotsData.Lot.QuantityInBag) AND ((Config.PremiumCount2 < (LotsData.Lot.QuantityInBag-10)) OR (Config.PremiumCount2 = LotsData.Lot.QuantityInBag))) THEN
			DropLocation := 1;
			NextState := eGoodULStaState.eDwell;
			PremiumFullCount := 0;
		ELSIF (Config.PremiumCount2 < LotsData.Lot.QuantityInBag) THEN
			DropLocation := 2;
			NextState := eGoodULStaState.eDwell;
			PremiumFullCount := 0;
		ELSE
			PartsData.Status[VUT].Premium := FALSE;
			PartsData.Status[VUT].Good := TRUE;
			PremiumFullCount := PremiumFullCount + 1;
		END_IF
	END_IF
	
	IF (PartsData.Status[VUT].Good) THEN      /// remove this after Turnkey Debug
		IF (NOT LotsData.Lot.AutoBaggerEnabled) THEN
			DropLocation := 3;
			NextState := eGoodULStaState.eDwell;
		ELSIF ((Config.GoodCount1 < LotsData.Lot.QuantityInBag) AND ((Config.GoodCount2 < (LotsData.Lot.QuantityInBag-10)) OR (Config.GoodCount2 = LotsData.Lot.QuantityInBag))) THEN
			DropLocation := 3;
			NextState := eGoodULStaState.eDwell;
			GoodFullCount := 0;
		ELSIF (NOT (Config.GoodCount2 >= LotsData.Lot.QuantityInBag)) THEN
			DropLocation := 4;
			NextState := eGoodULStaState.eDwell;
			GoodFullCount := 0;
		ELSE
			PartsData.Status[VUT].Premium := FALSE;
			PartsData.Status[VUT].Good := FALSE;
			PartsData.Status[VUT].OverallStatus := ePartStatus.eReject;
			PartsData.Status[VUT].GoodUnload := FALSE;
			GoodFullCount := GoodFullCount + 1;
		END_IF	
	END_IF
    	
	IF (PartsData.Status[VUT].OverallStatus = ePartStatus.eReject) THEN
		NextState := eGoodULStaState.eAbandonCycle;
	END_IF	
	
	IF (GoodFullCount >= 5 OR PremiumFullCount >= 5) THEN
		Stations.fbCycleControl.StopRequested := TRUE;
		Status.AutoBaggerStatusMsg := 'AutoBagger: No drop location available.';
	END_IF
	

eGoodULStaState.eDwell:
    DwellTimer(IN:=GVL_IO.UL_XBarrelPresent, PT := T#50MS);  /// Need to add Part Data to get this status to find if part needs to be rejected
	IF (DwellTimer.Q) THEN		
        NextState := eGoodULStaState.eEngagePalletHoldDown;
		ResetDwellTimer();
		ResetStateTimer();
    END_IF
	StateTimer(IN:=TRUE, PT:= T#1S);
	IF (StateTimer.Q) THEN
		NextState := eGoodULStaState.eAbandonCycle;
		ResetStateTimer();
		ResetDwellTimer();
		//NextState := eGoodULStaState.eEngagePalletHoldDown;
	END_IF
	
 eGoodULStaState.eAbandonCycle:
 	Act_FreePalletHold();
	Act_FreePalletRelease();
	IF (IsPalletHoldDownFree() AND IsPalletReleaseFree()) THEN
		ResetDwellTimer();
        NextState := eGoodULStaState.eDepartVehicle;
		Stations.fbRoutePlanner.M_NotifyVehStaCmpl(StationIndex:= MM_CONST.GOOD_UNLOAD_STA, VehicleID := VUT);
		xTrigger:= FALSE;
	END_IF
	
   DwellTimer(IN:=TRUE, PT:= T#10S);
   IF (DwellTimer.Q) THEN
		ErrorReturnState := eGoodULStaState.eHPReset;		
		ResetDwellTimer();
		ResetStateTimer();		
        NextState := eGoodULStaState.eError;		
	END_IF
	
		
eGoodULStaState.eEngagePalletHoldDown:

	Act_EngagePalletHold();
	NextState := eGoodULStaState.ePalletHoldDownEngaged;;
	IF (IsPalletHoldDownEngaged()) THEN	 // speed up more, don't wait here
		NextState := eGoodULStaState.ePalletHoldDownEngaged;
        //NextState := eGoodULStaState.eAbandonCycle;		
	END_IF
	
eGoodULStaState.ePalletHoldDownEngaged:
	//NextState:= eGoodULStaState.ePalletReleaseExtend;
	NextState := eGoodULStaState.eHPMoveToPickFromTrack;
	ResetDwellTimer();
	ResetStateTimer();
	
eGoodULStaState.eHPMoveToPickFromTrack:
    SetPPSequence(SequenceNumb := 2); // Pick location    
	Act_MoveRotatorCenter(); // also move rotary while going down
   	DwellTimer(IN:= TRUE, PT:= T#20MS);
   	IF (DwellTimer.Q) THEN
	   GVL_IO.UL_YPP_StartSeq := TRUE;
	   ResetDwellTimer();
   END_IF
   StateTimer(IN:= GVL_IO.UL_YPP_StartSeq, PT:= T#20MS);
   IF (StateTimer.Q) THEN
	   NextState := eGoodULStaState.eHPAtPickFromTrack;
	   ResetDwellTimer();
	   ResetStateTimer();
   END_IF


eGoodULStaState.eHPAtPickFromTrack:
	IF (CurrPPLoc = 2 ) THEN
		//NextState:= eGoodULStaState.eHPCloseGrippers;
		NextState := eGoodULStaState.eHPMoveToRotaryCenter;
		ResetDwellTimer();
		GVL_IO.UL_YPP_StartSeq := FALSE;
	END_IF

		
   DwellTimer(IN:=TRUE, PT:= T#10S);
   IF (DwellTimer.Q) THEN
		ErrorReturnState := eGoodULStaState.eHPMoveToPickFromTrack;		
		ResetDwellTimer();
		ResetStateTimer();		
		GVL_IO.UL_YPP_StartSeq := TRUE;
        NextState := eGoodULStaState.eError;		
		Status.GoodULStatusMsg:= 'Unload: PP Not At Pick Location';
	END_IF
	
	
	
eGoodULStaState.eHPMoveToRotaryCenter:

	Act_MoveRotatorCenter();
	NextState := eGoodULStaState.eHPAtRotaryCenter;

eGoodULStaState.eHPAtRotaryCenter:

	 IF (IsRotatorCenter()) THEN
		//NextState := eGoodULStaState.eDepartVehicle;
		NextState:= eGoodULStaState.eHPCloseGrippers;
		ResetDwellTimer();
	END_IF
	
   DwellTimer(IN:=TRUE, PT:= T#10S);
   IF (DwellTimer.Q) THEN
		ErrorReturnState := eGoodULStaState.eHPMoveToRotaryCenter;		
		ResetDwellTimer();
		ResetStateTimer();	
        NextState := eGoodULStaState.eError;	
		
	END_IF
	

	
eGoodULStaState.eHPCloseGrippers:
	Act_CloseGrippers();
	//Act_EngagePalletRelease();
	IF (IsGripperClosed()) THEN
		//NextState := eGoodULStaState.eHPGrippersClosed;
		Act_EngagePalletRelease();
	END_IF
	
	//These three lines of code should be commented out to revert the sequence change
	IF (IsPalletReleaseEngaged() AND IsGripperClosed()) THEN
		NextState := eGoodULStaState.eHPGrippersClosed;
		ResetDwellTimer();
	END_IF
	
   DwellTimer(IN:=TRUE, PT:= T#10S);
   IF (DwellTimer.Q) THEN
		ErrorReturnState := eGoodULStaState.eHPCloseGrippers;		
		ResetDwellTimer();
		ResetStateTimer();	
        NextState := eGoodULStaState.eError;			
	END_IF


eGoodULStaState.eHPGrippersClosed: //add logic here to decide which bagger location to go
	//NextState := eGoodULStaState.eHPSendToInitLocNext;
    IF (IsPalletHoldDownEngaged()) THEN	 
      NextState:= eGoodULStaState.ePalletReleaseExtend;
	  ResetDwellTimer();
	END_IF 
	
   DwellTimer(IN:=TRUE, PT:= T#10S);
   IF (DwellTimer.Q) THEN
		ErrorReturnState := eGoodULStaState.eEngagePalletHoldDown;		
		ResetDwellTimer();
		ResetStateTimer();	
        NextState := eGoodULStaState.eError;			
	END_IF



eGoodULStaState.ePalletReleaseExtend:

	Act_EngagePalletRelease();
	IF (IsPalletReleaseEngaged()) THEN
		   NextState := eGoodULStaState.ePalletReleaseExtended;		   
		   ResetDwellTimer();
	END_IF

eGoodULStaState.ePalletReleaseExtended:
	DwellTimer(IN:= TRUE, PT := T#100MS);
	IF (DwellTimer.Q) THEN 
		NextState := eGoodULStaState.eHPSendToInitLocNext;
		ResetDwellTimer();
	END_IF
  

eGoodULStaState.eHPSendToInitLocNext:
   // we have to set Seq 1 as InitLoc ( Up at Pick Location). Also, Input bits will corresponding to the sequence 
   SetPPSequence(SequenceNumb := 1);
   DwellTimer(IN:= TRUE, PT:= T#20MS);
   IF (DwellTimer.Q) THEN
	   GVL_IO.UL_YPP_StartSeq := TRUE;
	   DwellTimer(IN:=FALSE);
   END_IF
   StateTimer(IN:= GVL_IO.UL_YPP_StartSeq, PT:= T#20MS);
   IF (StateTimer.Q) THEN
	   NextState := eGoodULStaState.eHPAtInitLocNext;
	   ResetDwellTimer();
	   ResetStateTimer();
   END_IF
 
eGoodULStaState.eHPAtInitLocNext:
	IF (CurrPPLoc = 1 ) THEN
		NextState:= eGoodULStaState.eReleasePalletHoldDown;		
		GVL_IO.UL_YPP_StartSeq := FALSE;
		UpdateLotData();
		UpdatePartData();		
		ResetDwellTimer();
	END_IF
	
			
   DwellTimer(IN:=TRUE, PT:= T#10S);
   IF (DwellTimer.Q) THEN
		ErrorReturnState := eGoodULStaState.eHPSendToInitLocNext;		
		ResetDwellTimer();
		ResetStateTimer();		
		GVL_IO.UL_YPP_StartSeq := TRUE;
        NextState := eGoodULStaState.eError;		
		Status.GoodULStatusMsg:= 'Unload: PP Not At Init Location Next';
	END_IF

	
eGoodULStaState.eReleasePalletHoldDown:
	Act_FreePalletRelease();
	//Act_FreePalletHold();
	NextState := eGoodULStaState.eHPMoveToPlaceInBagLoc1; //eGoodULStaState.ePalletHoldDownReleased;

	
eGoodULStaState.eHPMoveToPlaceInBagLoc1:

	IF (DropLocation = 1 OR DropLocation = 3) THEN
		SetPPSequence(SequenceNumb := 3);
	ELSIF (DropLocation = 2 OR DropLocation = 4) THEN
		SetPPSequence(SequenceNumb := 4);
	ELSE
		Status.GoodULStatusMsg:= 'Unload: Problem with Pick & Place logic'; 
		NextState := eGoodULStaState.eUnknown; 
   	END_IF
	DwellTimer(IN:= TRUE, PT:= T#20MS);
   	IF (DwellTimer.Q) THEN
	   GVL_IO.UL_YPP_StartSeq := TRUE;
	   DwellTimer(IN:=FALSE);
   END_IF
   StateTimer(IN:= GVL_IO.UL_YPP_StartSeq, PT:= T#20MS);
   IF (StateTimer.Q) THEN
	   NextState := eGoodULStaState.eHPAtPlaceinBagLoc1;
	   ResetDwellTimer();
	   ResetStateTimer();
	   IF (DropLocation = 1 OR DropLocation = 2) THEN
			Act_MoveRotatorRight();
		ELSE
	   		Act_MoveRotatorLeft();
		END_IF	  
   END_IF
   
 eGoodULStaState.eHPAtPlaceinBagLoc1:
	IF ((CurrPPLoc = 3 AND DropLocation = 1) OR 
		(CurrPPLoc = 3 AND DropLocation = 3) OR
        (CurrPPLoc = 4 AND DropLocation = 2) OR 
		(CurrPPLoc = 4 AND DropLocation = 4)) THEN		
		IF (DropLocation = 1 OR DropLocation = 2) THEN
			Act_MoveRotatorRight();
		ELSE
	   		Act_MoveRotatorLeft();
		END_IF
		NextState:= eGoodULStaState.ePalletHoldDownReleased; //
		Act_FreePalletHold(); // we moved this so that pallet release is down before hold down. Maybe helps in jams
		GVL_IO.UL_YPP_StartSeq := FALSE;
		StateTimer(IN:=FALSE);
		ResetDwellTimer();
	END_IF
	
   DwellTimer(IN:=TRUE, PT:= T#10S);
   IF (DwellTimer.Q) THEN
		ErrorReturnState := eGoodULStaState.eHPMoveToPlaceInBagLoc1;		
		ResetDwellTimer();
		ResetStateTimer();		
		GVL_IO.UL_YPP_StartSeq := FALSE;
        NextState := eGoodULStaState.eError;		
		Status.GoodULStatusMsg:= 'Unload: PP Not At Init Location Next';
	END_IF


eGoodULStaState.ePalletHoldDownReleased: // release the Pallet Release At the same time ? 

	IF ( IsPalletHoldDownFree() AND IsPalletReleaseFree()) THEN
	 	 NextState:= eGoodULStaState.eAtCorrectRotaryLoc;
	 	Stations.fbRoutePlanner.M_NotifyVehStaCmpl(StationIndex:= MM_CONST.GOOD_UNLOAD_STA, VehicleID := VUT);
		xTrigger := FALSE;
		ResetDwellTimer();
    END_IF	
	
	DwellTimer(IN:=TRUE, PT:= T#10S);
   IF (DwellTimer.Q) THEN
		ErrorReturnState := eGoodULStaState.eHPAtPlaceinBagLoc1;		
		ResetDwellTimer();
		ResetStateTimer();		
        NextState := eGoodULStaState.eError;	
	END_IF

eGoodULStaState.eAtCorrectRotaryLoc:
    IF (DropLocation = 1 OR DropLocation = 2) THEN
		IF (IsRotatorRight()) THEN
			NextState := eGoodULStaState.eHPOpenGrippers;
			ResetDwellTimer();
		END_IF
	ELSE
    	IF (IsRotatorLeft()) THEN
			NextState := eGoodULStaState.eHPOpenGrippers;
			ResetDwellTimer();
		END_IF
    END_IF

    DwellTimer(IN:=TRUE, PT:= T#10S);
   IF (DwellTimer.Q) THEN
		ErrorReturnState := eGoodULStaState.eHPMoveToPlaceInBagLoc1;		
		ResetDwellTimer();
		ResetStateTimer();		
        NextState := eGoodULStaState.eError;	
	END_IF 	

	
	
eGoodULStaState.eHPOpenGrippers:
	Act_OpenGrippers();
	DwellTimer(IN:=TRUE, PT:= T#30MS);
	IF (DwellTimer.Q) THEN
		NextState := eGoodULStaState.eHPGrippersOpen;
		DwellTimer(IN:=FALSE);
	END_IF

eGoodULStaState.eHPGrippersOpen: //add logic here to increment parts in bag counter. //Done
	IF (IsGripperOpen()) THEN
		DwellTimer(IN:=TRUE, PT:= GripperOpenTimer);
		IF (DwellTimer.Q) THEN
			IF (DropLocation = 1 AND LotsData.Lot.AutoBaggerEnabled) THEN
				Config.PremiumCount1 := Config.PremiumCount1 + 1;
			ELSIF (DropLocation = 2 AND LotsData.Lot.AutoBaggerEnabled) THEN
				Config.PremiumCount2 := Config.PremiumCount2 + 1;
			ELSIF (DropLocation = 3 AND LotsData.Lot.AutoBaggerEnabled) THEN
				Config.GoodCount1 := Config.GoodCount1 + 1;
			ELSIF (DropLocation = 4 AND LotsData.Lot.AutoBaggerEnabled) THEN
				Config.GoodCount2 := Config.GoodCount2 + 1;
			END_IF
			NextState := eGoodULStaState.eHPSendToInitLocAfterDrop; //eGoodULStaState.eMoveRotaryRight;	
			DwellTimer(IN:=FALSE);
		END_IF         
	END_IF
	IF (xTrigger) THEN                                /// this is from the next vehicle coming in 
		Act_EngagePalletHold();
        IF (IsPalletHoldDownEngaged()) THEN
			;//Act_EngagePalletRelease();
		END_IF 
	END_IF
	
eGoodULStaState.eHPSendToInitLocAfterDrop:

   // we have to set Seq 1 as InitLoc ( Up at Pick Location). Also, Input bits will corresponding to the sequence 
  SetPPSequence(SequenceNumb := 1);
   DwellTimer(IN:= TRUE, PT:= T#20MS);
   IF (DwellTimer.Q) THEN
	   GVL_IO.UL_YPP_StartSeq := TRUE;
	   DwellTimer(IN:=FALSE);
   END_IF
   StateTimer(IN:= GVL_IO.UL_YPP_StartSeq, PT:= T#20MS);
   IF (StateTimer.Q) THEN
	   NextState := eGoodULStaState.eHPAtInitLocAfterDrop;//eGoodULStaState.eCheckRotaryAtRight;
       ResetDwellTimer(); 
   END_IF


eGoodULStaState.eHPAtInitLocAfterDrop:

	IF (CurrPPLoc = 1 ) THEN
		//NextState:= eGoodULStaState.eHPMoveToRotaryCenter;
		NextState := eGoodULStaState.eDepartVehicle;
		GVL_IO.UL_YPP_StartSeq := FALSE;
	END_IF

	
	IF (xTrigger) THEN                                /// this is from the next vehicle coming in 
		Act_EngagePalletHold();
        IF (IsPalletHoldDownEngaged()) THEN
	//		Act_EngagePalletRelease();
		END_IF 
	END_IF
	
	DwellTimer(IN:=TRUE, PT:= T#10S);
   IF (DwellTimer.Q) THEN
		ErrorReturnState := eGoodULStaState.eHPMoveToPlaceInBagLoc1;		
		ResetDwellTimer();
		ResetStateTimer();		
		GVL_IO.UL_YPP_StartSeq := FALSE;
        NextState := eGoodULStaState.eError;		
		Status.GoodULStatusMsg:= 'Unload: PP Not At Init Location After Drop';
	END_IF


(*	
	IF (xTrigger) THEN                                /// this is from the next vehicle coming in 
		Act_EngagePalletHold();
        IF (IsPalletHoldDownEngaged()) THEN
			Act_EngagePalletRelease();
		END_IF 
	END_IF
*)
eGoodULStaState.eDepartVehicle:

	IF (Stations.fbCycleControl.StopRequested) THEN
		NextState := eGoodULStaState.eStopActive;
	ELSE
		NextState := eGoodULStaState.eWaitForVehicleTrigger;
		DwellTimer(IN:=FALSE);
	END_IF

eGoodULStaState.eStopActive:
	IF (NOT Stations.fbCycleControl.StopRequested) THEN
		NextState := eGoodULStaState.eHPReady;
	END_IF
		

	
eGoodULStaState.eError:
	IF (GVL_IO.MC_XStartPB) THEN
		NextState := ErrorReturnState;
		ErrorReturnState := eGoodULStaState.eUnknown;
	END_IF
   
	
eGoodULStaState.eHPMoveToPlaceInBagLoc2:

	GVL_IO.UL_YPP_BitA := FALSE;
 	GVL_IO.UL_YPP_BitB := FALSE;
  	GVL_IO.UL_YPP_BitC := TRUE;
   	DwellTimer(IN:= TRUE, PT:= T#30MS);
   	IF (DwellTimer.Q) THEN
	   GVL_IO.UL_YPP_StartSeq := TRUE;
	   DwellTimer(IN:=FALSE);
   END_IF
   StateTimer(IN:= GVL_IO.UL_YPP_StartSeq, PT:= T#30MS);
   IF (StateTimer.Q) THEN
	   NextState := eGoodULStaState.eHPAtPlaceinBagLoc1;
   END_IF


eGoodULStaState.eHPAtPlaceinBagLoc2:

	IF (NOT GVL_IO.UL_XPP_A1OUT AND  NOT GVL_IO.UL_XPP_A2OUT AND GVL_IO.UL_XPP_A3OUT) THEN
		NextState:= eGoodULStaState.eTurnToRotartyCorrectSide;
		GVL_IO.UL_YPP_StartSeq := FALSE;
	END_IF
	StateTimer(IN:=TRUE, PT:= T#10S); // give a message out every 10 seconds
	IF (StateTimer.Q) THEN
		Logging.fbEventMsg.SendEventMsg(MsgClass := TCEVENTCLASS_STATEINFO, EventID:= Logging.ID_UL_PPWaitMoveCmpl, SourceID:= Logging.SrcGoodULPOU);
		StateTimer(IN:=FALSE);
	END_IF

eGoodULStaState.eTurnToRotartyCorrectSide: //WARNING !! this state is no longer used//add logic here to decide which side to turn the Rotary towards // this state is no longer used
    IF (DropLocation = 1 OR DropLocation = 2) THEN
		Act_MoveRotatorRight();
	ELSE
	    Act_MoveRotatorLeft();
	END_IF
	NextState := eGoodULStaState.eAtCorrectRotaryLoc;


eGoodULStaState.eMoveRotaryRight:
	GVL_IO.UL_YRotatorCWBarrelLeftBin := FALSE;;
	GVL_IO.UL_YRotatorCCWBarrelRightBin := TRUE;

	NextState := eGoodULStaState.eHPSendToInitLocAfterDrop; 





   eGoodULStaState.eCheckRotaryAtRight:
	 IF (NOT GVL_IO.UL_XRotatorCenter AND NOT GVL_IO.UL_XRotatorCWBarrelLeftBin AND GVL_IO.UL_XRotatorCWBarrelRightBin) THEN
		NextState := eGoodULStaState.eReleasePalletHoldDown;
	END_IF
	P_TextModeWrite.WriteData := FALSE; // Don't know if this is needed
	DwellTimer(IN:=TRUE, PT:= T#10S); // give a message out every 10 seconds
	IF (DwellTimer.Q) THEN
		Logging.fbEventMsg.SendEventMsg(MsgClass := TCEVENTCLASS_STATEINFO, EventID:= Logging.ID_UL_CheckCylinders, SourceID:= Logging.SrcGoodULPOU);
		DwellTimer(IN:=FALSE);	
	END_IF
	StateTimer(IN:=TRUE, PT:= T#30S);  // if it is more than 10 seconds then we send the station into an unknown state and wait for operator to fix and hit start button again
	IF (StateTimer.Q) THEN
		Logging.fbEventMsg.SendEventMsg(MsgClass := TCEVENTCLASS_STATEINFO, EventID:= Logging.ID_UL_CheckCylinders, SourceID:= Logging.SrcGoodULPOU);
		StateTimer(IN:=FALSE);
		NextState := eGoodULStaState.eReleasePalletHoldDown; //move the vehicle out.. we need to notify the operator some kind of alarm here 
	END_IF 
	


	
END_CASE

IF (State <> NextState) THEN
	bFirst := TRUE;
	StateTimer(IN:=FALSE);
ELSE
	bFirst := FALSE;
END_IF

State := NextState;
AssignStationStatusForHMI();

ACTION Act_CloseGrippers:
	GVL_IO.UL_YGrippersClose := TRUE;  
	GVL_IO.UL_YGrippersOpen := FALSE;
END_ACTION

ACTION ACT_EnablePP:
GVL_IO.UL_YPP_Enable := TRUE;   // Disable Drive
GVL_IO.UL_YPP_Stop := FALSE;      // Set Drive to Stop
GVL_IO.UL_YPP_ResetAlarm := FALSE;  // Clear Other Drive Inputs
GVL_IO.UL_YPP_StartHoming := FALSE;
END_ACTION

ACTION Act_EngagePalletHold:
GVL_IO.UL_YPalletHoldDownExtend_Home := FALSE; //Raise PalletHold Down 
GVL_IO.UL_YPalletHoldDownRetract_Engage := TRUE;
END_ACTION

ACTION Act_EngagePalletRelease:
//GVL_IO.UL_YPalletReleaseExtend := TRUE;    //Lower Pallet Release
//GVL_IO.UL_YPalletReleaseRetract := FALSE;
END_ACTION

ACTION Act_FreePalletHold:
GVL_IO.UL_YPalletHoldDownExtend_Home := TRUE; //Raise PalletHold Down 
GVL_IO.UL_YPalletHoldDownRetract_Engage := FALSE;
END_ACTION

ACTION Act_FreePalletRelease:
//GVL_IO.UL_YPalletReleaseExtend := FALSE;    //Lower Pallet Release
//GVL_IO.UL_YPalletReleaseRetract := TRUE;
END_ACTION

ACTION Act_MoveRotatorCenter:
GVL_IO.UL_YRotatorCCWBarrelRightBin := TRUE; //Move Rotator to Center Location
GVL_IO.UL_YRotatorCWBarrelLeftBin := TRUE;// Move the Rotator to Center Location
END_ACTION

ACTION Act_MoveRotatorLeft:
GVL_IO.UL_YRotatorCCWBarrelRightBin := FALSE; //Move Rotator to Center Location
   GVL_IO.UL_YRotatorCWBarrelLeftBin := TRUE;// Move the Rotator to Center Location
END_ACTION

ACTION Act_MoveRotatorRight:
GVL_IO.UL_YRotatorCCWBarrelRightBin := TRUE; //Move Rotator to Center Location
GVL_IO.UL_YRotatorCWBarrelLeftBin := FALSE;// Move the Rotator to Center Location
END_ACTION

ACTION Act_OpenGrippers:
GVL_IO.UL_YGrippersClose := FALSE;  //Open grippers
GVL_IO.UL_YGrippersOpen := TRUE;
END_ACTION

ACTION Act_ResetPPIO:
	//PP fieldbus commands
	GVL_IO.UL_YPP_BitA := FALSE;   // Turn off selection bits
	GVL_IO.UL_YPP_BitB := FALSE;
	GVL_IO.UL_YPP_BitC := FALSE;
	GVL_IO.UL_YPP_Enable := FALSE;   // Disable Drive
	GVL_IO.UL_YPP_Stop := TRUE;      // Set Drive to Stop
	GVL_IO.UL_YPP_ResetAlarm := FALSE;  // Clear Other Drive Inputs
	GVL_IO.UL_YPP_StartHoming := FALSE;
	GVL_IO.UL_YPP_StartSeq := FALSE;
END_ACTION

METHOD PUBLIC AssignStationStatusForHMI : BOOL
VAR_INPUT
END_VAR
Status.StationsState[MM_CONST.GOOD_UNLOAD_STA_HMI_STATE] := State;
IF (NOT LotsData.Lot.GoodUnloadEnabled) THEN
	Status.StationStauts[MM_CONST.GOOD_UNLOAD_STA_HMI_STATE] := OverallStationStatus.eDisabled;
ELSE	
	CASE State OF
	eGoodULStaState.eUnknown,eGoodULStaState.eError:
		Status.StationStauts[MM_CONST.GOOD_UNLOAD_STA_HMI_STATE] := OverallStationStatus.eError;
    
    eGoodULStaState.eInit,eGoodULStaState.eHoming,
	eGoodULStaState.eHPReset,eGoodULStaState.eHPCheckEnabled,eGoodULStaState.eHPSendHome,
	eGoodULStaState.eHPHomed,eGoodULStaState.eHPSendToInitLoc, eGoodULStaState.eHPAtInitLoc,
	eGoodULStaState.eHPReady:
	     Status.StationStauts[MM_CONST.GOOD_UNLOAD_STA_HMI_STATE] := OverallStationStatus.eHoming;
	
   	eGoodULStaState.eWaitForVehicleTrigger:
	     Status.StationStauts[MM_CONST.GOOD_UNLOAD_STA_HMI_STATE] := OverallStationStatus.eWaitingForParts;
		 
	eGoodULStaState.eDwell,
	eGoodULStaState.eEngagePalletHoldDown,
	eGoodULStaState.ePalletHoldDownEngaged,
	eGoodULStaState.ePalletReleaseExtend,
	eGoodULStaState.ePalletReleaseExtended,
	eGoodULStaState.eHPMoveToRotaryCenter,
	eGoodULStaState.eHPAtRotaryCenter,
	eGoodULStaState.eHPMoveToPickFromTrack,
	eGoodULStaState.eHPAtPickFromTrack,
	eGoodULStaState.eHPCloseGrippers,
	eGoodULStaState.eHPGrippersClosed,
	eGoodULStaState.eHPSendToInitLocNext,
	eGoodULStaState.eHPAtInitLocNext,
	eGoodULStaState.eHPMoveToPlaceInBagLoc1,
	eGoodULStaState.eHPMoveToPlaceInBagLoc2,
	eGoodULStaState.eHPAtPlaceinBagLoc1,
	eGoodULStaState.eHPAtPlaceinBagLoc2,
	eGoodULStaState.eTurnToRotartyCorrectSide,
	eGoodULStaState.eAtCorrectRotaryLoc,
	eGoodULStaState.eHPOpenGrippers,
	eGoodULStaState.eHPGrippersOpen,	
	eGoodULStaState.eMoveRotaryRight,
	eGoodULStaState.eCheckRotaryAtRight,
	eGoodULStaState.eReleasePalletHoldDown,
	eGoodULStaState.eHPSendToInitLocAfterDrop,
	eGoodULStaState.ePalletHoldDownReleased,
    eGoodULStaState.eHPAtInitLocAfterDrop:
	    Status.StationStauts[MM_CONST.GOOD_UNLOAD_STA_HMI_STATE] := OverallStationStatus.eRunning;
	
	eGoodULStaState.eStopActive:
	    Status.StationStauts[MM_CONST.GOOD_UNLOAD_STA_HMI_STATE] := OverallStationStatus.eCycleStop;
	ELSE;
	END_CASE
END_IF
END_METHOD

METHOD PUBLIC ClearVehicleTrigger : BOOL
VAR_INPUT
END_VAR
xTrigger := FALSE;
END_METHOD

METHOD PUBLIC GetPPLocation : BOOL
VAR_INPUT
END_VAR
VAR_OUTPUT
	Location : BYTE;
END_VAR
Location.0 := GVL_IO.UL_XPP_A1OUT;
Location.1 := GVL_IO.UL_XPP_A2OUT;
Location.2 := GVL_IO.UL_XPP_A3OUT;
END_METHOD

METHOD PUBLIC IsFaulted : BOOL
VAR_INPUT
END_VAR
IsFaulted := (State = eGoodULStaState.eUnknown OR State = eGoodULStaState.eError);
END_METHOD

METHOD PUBLIC IsGripperClosed : BOOL
VAR_INPUT
END_VAR
IsGripperClosed := (NOT GVL_IO.UL_XGrippersOpened (*AND GVL_IO.UL_XGrippersClosed*)); 
IF(NOT IsGripperClosed) THEN
	Status.GoodULStatusMsg:= 'Unload: Check Gripper Sensors';
END_IF
END_METHOD

METHOD PUBLIC IsGripperOpen : BOOL
VAR_INPUT
END_VAR
IsGripperOpen := (GVL_IO.UL_XGrippersOpened AND NOT GVL_IO.UL_XGrippersClosed); 
IF(NOT IsGripperOpen) THEN
	Status.GoodULStatusMsg:= 'Unload: Check Gripper Sensors';
END_IF
END_METHOD

METHOD PUBLIC IsPalletHoldDownEngaged : BOOL
VAR_INPUT
END_VAR
IsPalletHoldDownEngaged := (NOT GVL_IO.UL_XPalletHoldDownExtended_Home AND GVL_IO.UL_XPalletHoldDownRetracted_Engaged);
IF (NOT IsPalletHoldDownEngaged) THEN Status.GoodULStatusMsg := 'Failed to Engage Pallet HoldDown Sensors'; END_IF
END_METHOD

METHOD PUBLIC IsPalletHoldDownFree : BOOL
VAR_INPUT
END_VAR
IsPalletHoldDownFree := (GVL_IO.UL_XPalletHoldDownExtended_Home AND NOT GVL_IO.UL_XPalletHoldDownRetracted_Engaged);
IF (NOT IsPalletHoldDownFree) THEN Status.GoodULStatusMsg := 'Failed to Release Pallet HoldDown Sensors'; END_IF
END_METHOD

METHOD PUBLIC IsPalletReleaseEngaged : BOOL
VAR_INPUT
END_VAR
IsPalletReleaseEngaged := TRUE; // The new Pallet Design doesn't require Pallet Release to be Engaged
//IsPalletReleaseEngaged := (NOT GVL_IO.UL_XPalletReleaseHome AND GVL_IO.UL_XPalletReleaseExtended);
//IF (NOT IsPalletReleaseEngaged) THEN Status.GoodULStatusMsg := 'Unload: Check Pallet Release Sensors'; END_IF
END_METHOD

METHOD PUBLIC IsPalletReleaseFree : BOOL
VAR_INPUT
END_VAR
IsPalletReleaseFree := TRUE; // new Pallet Design doesn't require Pallet Release Engage to be Extended
//IsPalletReleaseFree := (GVL_IO.UL_XPalletReleaseHome AND NOT GVL_IO.UL_XPalletReleaseExtended);
//IF (NOT IsPalletReleaseFree) THEN Status.GoodULStatusMsg := 'Unload: Check Pallet Release Sensors'; END_IF
END_METHOD

METHOD PUBLIC IsRotatorCenter : BOOL
VAR_INPUT
END_VAR
IsRotatorCenter := (GVL_IO.UL_XRotatorCenter AND NOT GVL_IO.UL_XRotatorCWBarrelLeftBin AND NOT GVL_IO.UL_XRotatorCWBarrelRightBin);
IF (NOT IsRotatorCenter) THEN Status.GoodULStatusMsg := 'Not At Center Check Rotator Sensor'; END_IF
END_METHOD

METHOD PUBLIC IsRotatorLeft : BOOL
VAR_INPUT
END_VAR
IsRotatorLeft := (NOT GVL_IO.UL_XRotatorCenter AND GVL_IO.UL_XRotatorCWBarrelLeftBin AND NOT GVL_IO.UL_XRotatorCWBarrelRightBin);
IF (NOT IsRotatorLeft) THEN Status.GoodULStatusMsg := 'Not At Left Check Rotator Sensor'; END_IF
END_METHOD

METHOD PUBLIC IsRotatorRight : BOOL
VAR_INPUT
END_VAR
IsRotatorRight := (NOT GVL_IO.UL_XRotatorCenter AND NOT GVL_IO.UL_XRotatorCWBarrelLeftBin AND GVL_IO.UL_XRotatorCWBarrelRightBin);
IF (NOT IsRotatorRight) THEN Status.GoodULStatusMsg := 'Not At Right, Check Rotator Sensor'; END_IF
END_METHOD

PROPERTY PUBLIC Ready : BOOL
GET
IF (LotsData.Lot.GoodUnloadEnabled) THEN
	Ready := (State = eGoodULStaState.eWaitForVehicleTrigger);
ELSE
	Ready := (State = eGoodULStaState.eDisabledReady);	
END_IF
END_GET
END_PROPERTY

ACTION ResetDwellTimer:
DwellTimer(IN:=FALSE);
END_ACTION

METHOD ResetState : BOOL
VAR_INPUT
END_VAR
	State := eGoodULStaState.eUnknown;
	NextState := eGoodULStaState.eUnknown;
END_METHOD

ACTION ResetStateTimer:
StateTimer(IN:=FALSE);
END_ACTION

METHOD PUBLIC SetPPSequence : BOOL
VAR_INPUT
	SequenceNumb : BYTE;
END_VAR
CASE SequenceNumb OF 
	0:
	   GVL_IO.UL_YPP_BitA := FALSE;
   	   GVL_IO.UL_YPP_BitB := FALSE;
   	   GVL_IO.UL_YPP_BitC := FALSE;
	1:
	   GVL_IO.UL_YPP_BitA := TRUE;
   	   GVL_IO.UL_YPP_BitB := FALSE;
   	   GVL_IO.UL_YPP_BitC := FALSE;
	2:
	   GVL_IO.UL_YPP_BitA := FALSE;
   	   GVL_IO.UL_YPP_BitB := TRUE;
   	   GVL_IO.UL_YPP_BitC := FALSE;
	3:
	   GVL_IO.UL_YPP_BitA := TRUE;
   	   GVL_IO.UL_YPP_BitB := TRUE;
   	   GVL_IO.UL_YPP_BitC := FALSE;
	4:
		GVL_IO.UL_YPP_BitA := FALSE;
   	    GVL_IO.UL_YPP_BitB := FALSE;
   	    GVL_IO.UL_YPP_BitC := TRUE;
	5:
	    GVL_IO.UL_YPP_BitA := TRUE;
   	   	GVL_IO.UL_YPP_BitB := FALSE;
   	   	GVL_IO.UL_YPP_BitC := TRUE;
	6: 
	    GVL_IO.UL_YPP_BitA := FALSE;
   	   	GVL_IO.UL_YPP_BitB := TRUE;
   	   	GVL_IO.UL_YPP_BitC := TRUE;
	7:
	    GVL_IO.UL_YPP_BitA := TRUE;
   	    GVL_IO.UL_YPP_BitB := TRUE;
   	    GVL_IO.UL_YPP_BitC := TRUE;
	ELSE;
			
END_CASE
END_METHOD

PROPERTY PUBLIC Trigger : BOOL
SET
xTrigger := Trigger;
END_SET
END_PROPERTY

METHOD PUBLIC UpdateLotData : BOOL
VAR_INPUT
END_VAR
IF (PartsData.Status[VUT].Premium) THEN
	LotsData.Lot.CavityCounts[PartsData.Status[VUT].CavityNumber].PremiumCount := LotsData.Lot.CavityCounts[PartsData.Status[VUT].CavityNumber].PremiumCount +1;
ELSIF (PartsData.Status[VUT].Good) THEN
 	LotsData.Lot.CavityCounts[PartsData.Status[VUT].CavityNumber].GoodCount := LotsData.Lot.CavityCounts[PartsData.Status[VUT].CavityNumber].GoodCount + 1;
END_IF
LotsData.Lot.CavityCounts[PartsData.Status[VUT].CavityNumber].TotalCount := LotsData.Lot.CavityCounts[PartsData.Status[VUT].CavityNumber].TotalCount + 1;
 // reject parts shouldn't get here. If this station rejects something (e.g. faults out) then it barrel will go to reject station.
END_METHOD

METHOD PUBLIC UpdatePartData : BOOL
VAR_INPUT
END_VAR
PartsData.Status[VUT].UnloadTime := SYSTEMTIME_TO_STRING(Logging.fbCurrTime.systemTime);
PartsData.Status[VUT].OverallStatus := ePartStatus.eEmpty;
PartsData.Status[VUT].GoodUnload := TRUE;

// we will write data to CSV file over here 
IF (P_TextModeWrite.CurrWriteStep = 0) THEN 
	P_TextModeWrite.VehicleID := VUT;
	P_TextModeWrite.WriteData := TRUE;
END_IF
END_METHOD

PROPERTY PUBLIC VehicleUnderTest : BYTE
GET
VehicleUnderTest := VUT;
END_GET
SET
VUT := VehicleUnderTest;
END_SET
END_PROPERTY

END_FUNCTION_BLOCK

// ---- POUs/AutoBagger.TcPOU
FUNCTION_BLOCK AutoBagger
VAR_INPUT
END_VAR
VAR_OUTPUT
END_VAR
VAR
	State : eAutoBaggerState := eAutoBaggerState.eUnknown;
	NextState : eAutoBaggerState := eAutoBaggerState.eUnknown;
	ErrorReturnState: eAutoBaggerState := eAutoBaggerState.eUnknown;
	DwellTimer : TON;
	StateTimer : TON;		
	ActiveChute : BYTE;
	bFirst : BOOL := FALSE;
	stopRequested : BOOL := FALSE;
	ShakeAttempts :BYTE :=0;
	MaxShakeAttempts: BYTE := 2;
	
END_VAR

IF (NOT LotsData.Lot.AutoBaggerEnabled) THEN
	NextState := eAutoBaggerState.eInit;
END_IF
//   If valve is changed so that the chutes remain closed on E-Stop then comment out the block below by removing the //
//(*
IF (GVL_IO.MachineEStopped) THEN 
	Config.PremiumCount1 := 0;
	Config.PremiumCount2 := 0;
	Config.GoodCount1 := 0;
	Config.GoodCount2 := 0;
END_IF
//*)   
//  If valve is changed so that the chutes remain closed on E-Stop then remove the slash on the line above 

CASE State OF

eAutoBaggerState.eUnknown:
   IF (GVL_IO.MC_XStartPB AND GVL_IO.MC_XAirPressureOK AND GVL_IO.MC_NotEStopped) THEN // wait for start button when powered up or PLC program restarted
		NextState := eAutoBaggerState.eInit;	   
   END_IF

eAutoBaggerState.eInit:
	StateTimer(IN:=TRUE, PT:= T#10S);
	
	IF (NOT LotsData.Lot.AutoBaggerEnabled) THEN
		Act_OpenGoodChute1();
		Act_OpenGoodChute2();
		Act_OpenPremiumChute1();
		Act_OpenPremiumChute2();		
		Status.AutoBaggerStatusMsg := 'Bagger Disabled';
		StateTimer(IN:=FALSE);
		Act_TriggerBaggerOFF();
	END_IF
	
	IF (LotsData.Lot.AutoBaggerEnabled) THEN
		Act_CloseTrapDoor();
		Act_TriggerBaggerOFF();
		IF (ChuteClosed) THEN    //All Chutes are closed 
			NextState := eAutoBaggerState.eCheckWaitingLabel;
			Status.AutoBaggerStatusMsg := '';
			StateTimer(IN:=FALSE);
		END_IF
	END_IF 
	
	IF(StateTimer.Q AND LotsData.Lot.AutoBaggerEnabled AND NOT ChuteClosed) THEN
		NextState := eAutoBaggerState.eError;
		ErrorReturnState := eAutoBaggerState.eInit; 
		Status.AutoBaggerStatusMsg := 'AutoBagger: Unable to Close Chutes, Fix & Press START ';
		StateTimer(IN:=FALSE);
	END_IF

eAutoBaggerState.eCheckWaitingLabel: //checking to see if Step 1 in document is OK i.e. Not Faulted, Waiting for Label and Not Ready for filler
	StateTimer(IN:=TRUE, PT:= T#10S);
	IF (IsBaggerWaitingForLabel() AND IsBaggerOK_NotFaulted() (*AND IsBagClosed()*)) THEN
		NextState := eAutoBaggerState.eReady;
		StateTimer(IN:=FALSE);
	END_IF
	IF(StateTimer.Q ) THEN
		NextState := eAutoBaggerState.eError;
		ErrorReturnState := eAutoBaggerState.eCheckWaitingLabel;
		StateTimer(IN:=FALSE);
	END_IF

//Wait for one chute to fill up
eAutoBaggerState.eReady:
	Act_CloseTrapDoor();
	IF (Config.PremiumCount1 = LotsData.Lot.QuantityInBag) THEN
		ActiveChute := 1;
		NextState := eAutoBaggerState.eSendLabel;
	ELSIF (Config.PremiumCount2 = LotsData.Lot.QuantityInBag) THEN
		ActiveChute := 2;
		NextState := eAutoBaggerState.eSendLabel;
	ELSIF (Config.GoodCount1 = LotsData.Lot.QuantityInBag) THEN
		ActiveChute := 3;
		NextState := eAutoBaggerState.eSendLabel;
	ELSIF (Config.GoodCount2 = LotsData.Lot.QuantityInBag) THEN
		ActiveChute := 4;
		NextState := eAutoBaggerState.eSendLabel;
	END_IF
	
	
//send label and print command
eAutoBaggerState.eSendLabel:
	
	IF(ActiveChute = 1 OR ActiveChute = 2) THEN //Send Premium label
		M_SendLabel(TRUE);		
	ELSE
		M_SendLabel(FALSE);		
	END_IF
	NextState := eAutoBaggerState.eWaitForBagOpen;	


eAutoBaggerState.eWaitForBagOpen:
	StateTimer(IN:=TRUE, PT := T#10S);
	IF (IsBaggerLabelPrinted() AND IsBaggerOK_NotFaulted() AND IsBaggerOpenWaitingforParts()) THEN
		NextState := eAutoBaggerState.eDropParts;
		ShakeAttempts:=0;
		StateTimer(IN:=FALSE);
	END_IF
	
	IF(StateTimer.Q ) THEN
		NextState := eAutoBaggerState.eError;
		ErrorReturnState := eAutoBaggerState.eHandleBagOpenError;
		StateTimer(IN:=FALSE);
	END_IF
	
eAutoBaggerState.eHandleBagOpenError:

IF (IsBaggerWaitingForLabel()) THEN
	NextState := eAutoBaggerState.eSendLabel;
ELSIF (IsBaggerLabelPrinted() AND IsBaggerOK_NotFaulted() AND IsBaggerOpenWaitingforParts()) THEN
		NextState := eAutoBaggerState.eDropParts;
ELSE
	NextState := eAutoBaggerState.eError;
	ErrorReturnState := eAutoBaggerState.eHandleBagOpenError;
	StateTimer(IN:=FALSE);		
END_IF
		

eAutoBaggerState.eDropParts:
//open trap door for (chute)
	StateTimer(IN:=TRUE, PT:= T#20S);
	IF (ActiveChute = 3) THEN//Prioritize Good chutes because Premium can go into good, so we waste less.  
		Act_OpenGoodChute1();
		DwellTimer(IN:=TRUE, PT:= T#4S);
	ELSIF (ActiveChute = 4) THEN
		Act_OpenGoodChute2();
		DwellTimer(IN:=TRUE, PT:= T#4S);
	ELSIF (ActiveChute = 1) THEN
		Act_OpenPremiumChute1();
		DwellTimer(IN:=TRUE, PT:= T#4S);
	ELSIF (ActiveChute = 2) THEN
		Act_OpenPremiumChute2();
		DwellTimer(IN:=TRUE, PT:= T#4S);
	END_IF

//wait long enough for parts to drop, then move to next state
	IF (DwellTimer.Q AND ChuteOpen AND NOT ChuteClosed) THEN
		NextState := eAutoBaggerState.eHalfCloseTrapDoor;
		/// If you want to skip the trap door double cycle, then uncomment the line below and login->online change, check update boot project
		//NextState := eAutoBaggerState.eCloseTrapDoor;   
		DwellTimer(IN:=FALSE);
		StateTimer(IN:=FALSE);
	END_IF	
	
	IF (StateTimer.Q AND NOT ChuteOpen) THEN
		NextState := eAutoBaggerState.eError;
		ErrorReturnState := eAutoBaggerState.eDropParts;
		Status.AutoBaggerStatusMsg := 'AutoBagger: Unable to open chute door. Fix then hit START';
		StateTimer(IN:=FALSE);
		DwellTimer(IN:=FALSE);
	END_IF

eAutoBaggerState.eHalfCloseTrapDoor:

    Act_CloseTrapDoor();
	StateTimer(IN:=TRUE, PT:= T#1000MS);
	IF (StateTimer.Q) THEN
		NextState := eAutoBaggerState.eOpenTrapDoorFinal;		
		StateTimer(IN:=FALSE);
		DwellTimer(IN:=FALSE);
		ShakeAttempts := ShakeAttempts + 1;
	END_IF
	
eAutoBaggerState.eOpenTrapDoorFinal:
//open trap door FOR (chute)
	StateTimer(IN:=TRUE, PT:= T#20S);
	IF (ActiveChute = 3) THEN//Prioritize Good chutes because Premium can go into good, so we waste less.  
		Act_OpenGoodChute1();
		DwellTimer(IN:=TRUE, PT:= T#3S);
	ELSIF (ActiveChute = 4) THEN
		Act_OpenGoodChute2();
		DwellTimer(IN:=TRUE, PT:= T#3S);
	ELSIF (ActiveChute = 1) THEN
		Act_OpenPremiumChute1();
		DwellTimer(IN:=TRUE, PT:= T#3S);
	ELSIF (ActiveChute = 2) THEN
		Act_OpenPremiumChute2();
		DwellTimer(IN:=TRUE, PT:= T#3S);
	END_IF

//wait long enough for parts to drop, then move to next state
	IF (DwellTimer.Q AND ChuteOpen AND NOT ChuteClosed) THEN
		NextState := eAutoBaggerState.eCloseTrapDoor;
		DwellTimer(IN:=FALSE);
		StateTimer(IN:=FALSE);
	END_IF	
	
	IF (StateTimer.Q AND NOT ChuteOpen) THEN
		NextState := eAutoBaggerState.eError;
		ErrorReturnState := eAutoBaggerState.eDropParts;
		Status.AutoBaggerStatusMsg := 'AutoBagger: Unable to open chute door. Fix then hit START';
		StateTimer(IN:=FALSE);
		DwellTimer(IN:=FALSE);
	END_IF
	

	
eAutoBaggerState.eCloseTrapDoor:
	Act_CloseTrapDoor();
	StateTimer(IN:=TRUE, PT:= T#10S);
	IF (ChuteClosed AND NOT ChuteOpen) THEN
		NextState := eAutoBaggerState.eTriggerBagger;
		StateTimer(IN:=FALSE);
		
	END_IF	
	
	IF (StateTimer.Q AND NOT ChuteClosed) THEN
		IF (ShakeAttempts < MaxShakeAttempts) THEN
			NextState := eAutoBaggerState.eHalfCloseTrapDoor;
		ELSE
			Status.AutoBaggerStatusMsg := 'Chute door CANNOT close. Clear jams, then hit START';
			NextState := eAutoBaggerState.eError;
			ErrorReturnState := eAutoBaggerState.eCloseTrapDoor;
			StateTimer(IN:=FALSE);
			DwellTimer(IN:=FALSE);
		END_IF
	END_IF

	

eAutoBaggerState.eTriggerBagger:
	ShakeAttempts := 0;
	ACT_TriggerBaggerON();
	DwellTimer(IN:=TRUE, PT:= T#500MS);
	
	IF (DwellTimer.Q) THEN
		NextState := eAutoBaggerState.eWaitforBaggingStart;
		IF (ActiveChute = 1) THEN
			Config.PremiumCount1 := 0;
		ELSIF (ActiveChute = 2) THEN
			Config.PremiumCount2 := 0;
		ELSIF (ActiveChute = 3) THEN
			Config.GoodCount1 := 0;
		ELSIF (ActiveChute = 4) THEN
			Config.GoodCount2 := 0;
		END_IF
		DwellTimer(IN:=FALSE);
	END_IF	
	
eAutoBaggerState.eWaitforBaggingStart:
		StateTimer(IN:=TRUE, PT:= T#10S);
		IF (NOT IsBaggerOpenWaitingforParts()) THEN
			ACT_TriggerBaggerOFF();
			NextState := eAutoBaggerState.eWaitforBaggingComplete;
		END_IF
		
	IF (StateTimer.Q AND IsBaggerOpenWaitingforParts()) THEN
		Status.AutoBaggerStatusMsg := 'Autobagger DIDNT start bagging. Fix Error & hit START';
		NextState := eAutoBaggerState.eError;
		ErrorReturnState := eAutoBaggerState.eTriggerBagger;
		IF (IsBaggerWaitingForLabel()) THEN 
			ErrorReturnState := eAutoBaggerState.eSendLabel;
		END_IF
		ACT_TriggerBaggerOFF();
		StateTimer(IN:=FALSE);
		DwellTimer(IN:=FALSE);
	END_IF	
		
eAutoBaggerState.eWaitForBaggingComplete:
	StateTimer(IN:=TRUE, PT := T#20S);
	IF (IsBaggerWaitingForLabel()) THEN
		NextState := eAutoBaggerState.eReady;
		StateTimer(IN:=FALSE);
	END_IF
	
	IF (StateTimer.Q AND NOT IsBaggerWaitingForLabel()) THEN
		Status.AutoBaggerStatusMsg := 'Autobagger DIDNT complete bagging. Fix Error & hit START';
		NextState := eAutoBaggerState.eError;
		ErrorReturnState := eAutoBaggerState.eTriggerBagger;
		IF (IsBaggerWaitingForLabel()) THEN 
			ErrorReturnState := eAutoBaggerState.eSendLabel;
		END_IF
		IF (NOT IsBaggerOK_NotFaulted()) THEN
			ErrorReturnState := eAutoBaggerState.eInit;
		END_IF
		ACT_TriggerBaggerOFF();
		StateTimer(IN:=FALSE);
		DwellTimer(IN:=FALSE);
	END_IF	

eAutoBaggerState.eError: 
			
	Status.StationStauts[MM_CONST.AUTOBAGGER_HMI_STATE] := OverallStationStatus.eError;
	IF (GVL_IO.MC_XStartPB) THEN
		NextState := ErrorReturnState;
		ErrorReturnState := eAutoBaggerState.eError;
	END_IF
	
END_CASE

//If any chute holds more parts than the maximum number, send station to Error.  
(*
IF(Config.GoodCount1 > LotsData.Lot.QuantityInBag OR Config.GoodCount1 > LotsData.Lot.QuantityInBag OR Config.GoodCount1 > LotsData.Lot.QuantityInBag OR Config.GoodCount1 > LotsData.Lot.QuantityInBag) THEN
	NextState := eAutoBaggerState.eError;
	ErrorReturnState := eAutoBaggerState.eInit;
	Status.AutoBaggerStatusMsg := 'Chute Count MAX. Open/Close Chute, Clear Count then HIT START';
END_IF
*)
IF (State <> NextState) THEN
	bFirst := TRUE;
	StateTimer(IN:=FALSE);
ELSE
	bFirst := FALSE;
END_IF

State := NextState;
AssignStationStatusForHMI();

ACTION Act_CloseTrapDoor:
GVL_IO.BG_YOpenChute1 := FALSE;
GVL_IO.BG_YOpenChute2 := FALSE;
GVL_IO.BG_YOpenChute3 := FALSE;
GVL_IO.BG_YOpenChute4 := FALSE;

GVL_IO.BG_YCloseChute1 := TRUE;
GVL_IO.BG_YCloseChute2 := TRUE;
GVL_IO.BG_YCloseChute3 := TRUE;
GVL_IO.BG_YCloseChute4 := TRUE;
END_ACTION

ACTION Act_OpenGoodChute1:
GVL_IO.BG_YOpenChute3 := TRUE;
GVL_IO.BG_YCloseChute3 := FALSE;
END_ACTION

ACTION Act_OpenGoodChute2:
GVL_IO.BG_YOpenChute4 := TRUE;
GVL_IO.BG_YCloseChute4 := FALSE;
END_ACTION

ACTION Act_OpenPremiumChute1:
GVL_IO.BG_YOpenChute1 := TRUE;
GVL_IO.BG_YCloseChute1 := FALSE;
END_ACTION

ACTION Act_OpenPremiumChute2:
GVL_IO.BG_YOpenChute2 := TRUE;
GVL_IO.BG_YCloseChute2 := FALSE;
END_ACTION

ACTION Act_OpenTrapDoor:
IF (ActiveChute = 1) THEN
	GVL_IO.BG_YOpenChute1 := TRUE;
	GVL_IO.BG_YCloseChute1 := FALSE;
ELSIF (ActiveChute = 2) THEN
	GVL_IO.BG_YOpenChute2 := TRUE;
	GVL_IO.BG_YCloseChute2 := FALSE;
ELSIF (ActiveChute = 3) THEN
	GVL_IO.BG_YOpenChute3 := TRUE;
	GVL_IO.BG_YCloseChute3 := FALSE;
ELSIF (ActiveChute = 4) THEN
	GVL_IO.BG_YOpenChute4 := TRUE;
	GVL_IO.BG_YCloseChute4 := FALSE;
END_IF
END_ACTION

ACTION ACT_TriggerBaggerOFF:
GVL_IO.BG_YFillerTrigger := FALSE;
END_ACTION

ACTION ACT_TriggerBaggerON:
GVL_IO.BG_YFillerTrigger := TRUE;
END_ACTION

METHOD AssignStationStatusForHMI : BOOL
VAR_INPUT
END_VAR
Status.StationsState[MM_CONST.AUTOBAGGER_HMI_STATE] := State;
IF (NOT LotsData.Lot.AutoBaggerEnabled) THEN
	Status.StationStauts[MM_CONST.AUTOBAGGER_HMI_STATE] := OverallStationStatus.eDisabled;
ELSE	
	CASE State OF
	eAutoBaggerState.eUnknown,eAutoBaggerState.eError, eAutoBaggerState.eDoorCannotOpen, eAutoBaggerState.eDoorCannotClose, eAutoBaggerState.eMissingBusySignal, eAutoBaggerState.eMissingBusySignal2, eAutoBaggerState.eMissingNotBusySignal: 
		Status.StationStauts[MM_CONST.AUTOBAGGER_HMI_STATE] := OverallStationStatus.eError;
		
	eAutoBaggerState.eInit:
	    Status.StationStauts[MM_CONST.AUTOBAGGER_HMI_STATE] := OverallStationStatus.eHoming;
	
    eAutoBaggerState.eWaitForBaggerNotBusy, eAutoBaggerState.eWaitForBaggerBusy:
	    Status.StationStauts[MM_CONST.AUTOBAGGER_HMI_STATE] := OverallStationStatus.eWarning;
	
	eAutoBaggerState.eReady:
	    Status.StationStauts[MM_CONST.AUTOBAGGER_HMI_STATE] := OverallStationStatus.eWaitingForParts;
		 
    eAutoBaggerState.eCloseTrapDoor, eAutoBaggerState.eHalfCloseTrapDoor, eAutoBaggerState.eOpenTrapDoorFinal, eAutoBaggerState.eDetachBag1, eAutoBaggerState.eDetachBag2, eAutoBaggerState.eDropParts,
	eAutoBaggerState.eFeederReadyReset1, eAutoBaggerState.eFeederReadyReset2, eAutoBaggerState.eSendLabel: 
	    Status.StationStauts[MM_CONST.AUTOBAGGER_HMI_STATE] := OverallStationStatus.eRunning;
		
		//Status.StationStauts[MM_CONST.AUTOBAGGER_HMI_STATE] := OverallStationStatus.eCycleStop;
    
    ELSE ;	
	END_CASE
END_IF
END_METHOD

PROPERTY ChuteClosed : BOOL
GET
IF (GVL_IO.BG_XChute1Closed AND GVL_IO.BG_XChute2Closed AND GVL_IO.BG_XChute3Closed AND GVL_IO.BG_XChute4Closed) THEN
	ChuteClosed := TRUE;
ELSE
	ChuteClosed := FALSE;
END_IF
END_GET
END_PROPERTY

PROPERTY ChuteOpen : BOOL
GET
CASE ActiveChute OF
	1:
	ChuteOpen := GVL_IO.BG_XChute1Open;
	
	2:
	ChuteOpen := GVL_IO.BG_XChute2Open;
	
	3:
	ChuteOpen := GVL_IO.BG_XChute3Open;
	
	4:
	ChuteOpen := GVL_IO.BG_XChute4Open;
	
END_CASE

//ChuteOpen := TRUE;
END_GET
END_PROPERTY

METHOD PUBLIC IsBagClosed : BOOL
VAR_INPUT
END_VAR
IsBagClosed := NOT GVL_IO.BG_XBaggerReadyForFiller;
IF (NOT IsBagClosed) THEN
	Status.AutoBaggerStatusMsg := 'Autobagger: Bag is NOT CLOSED';
END_IF
END_METHOD

METHOD PUBLIC IsBaggerLabelPrinted : BOOL
VAR_INPUT
END_VAR
IsBaggerLabelPrinted := NOT GVL_IO.BG_XBaggerWaitingForLabel;
IF (NOT IsBaggerLabelPrinted) THEN
	Status.AutoBaggerStatusMsg := 'Bagger Label Not Printed, Check Line Mode Bagger HMI & hit START';
END_IF
END_METHOD

METHOD PUBLIC IsBaggerOK_NotFaulted : BOOL
VAR_INPUT
END_VAR
IsBaggerOK_NotFaulted := GVL_IO.BG_XBaggerOKNoFault;
IF (NOT IsBaggerOK_NotFaulted) THEN
	Status.AutoBaggerStatusMsg := 'AutoBagger: Bagger Is Faulted, Clear Faults from Bagger HMI & hit START ';
END_IF
END_METHOD

METHOD PUBLIC IsBaggerOpenWaitingforParts : BOOL
VAR_INPUT
END_VAR
IsBaggerOpenWaitingforParts := GVL_IO.BG_XBaggerReadyForFiller;
IF (NOT IsBaggerOpenWaitingforParts) THEN
	Status.AutoBaggerStatusMsg := 'Cant Open bag, Check Bagger HMI & hit START';
END_IF
END_METHOD

METHOD PUBLIC IsBaggerWaitingForLabel : BOOL
VAR_INPUT
END_VAR
IsBaggerWaitingForLabel := GVL_IO.BG_XBaggerWaitingForLabel;
IF (NOT IsBaggerWaitingForLabel) THEN
	Status.AutoBaggerStatusMsg := 'Bagger Not Waiting For Label, Check Line Mode Bagger HMI & hit START';
END_IF
END_METHOD

METHOD PUBLIC IsBagsLowWarning : BOOL
VAR_INPUT
END_VAR
IsBagsLowWarning := GVL_IO.BG_XBagsLow;
IF (NOT IsBagsLowWarning) THEN
	Status.AutoBaggerStatusMsg := 'Bagger Low Bags Warning, Change Roll';
END_IF
END_METHOD

METHOD PUBLIC IsFaulted : BOOL
VAR_INPUT
END_VAR
IF (LotsData.Lot.AutoBaggerEnabled) THEN 
	IsFaulted := (State = eAutoBaggerState.eUnknown OR State = eAutoBaggerState.eError);
ELSE 
	IsFaulted := FALSE;
END_IF
END_METHOD

METHOD M_SendLabel : BOOL
VAR_INPUT
	isPremium : BOOL;
END_VAR
MAIN.fbEL6001.M_PrintLabel(isPremium);
END_METHOD

PROPERTY PUBLIC Ready : BOOL
GET
IF (LotsData.Lot.AutoBaggerEnabled) THEN
 	Ready := (State = eAutoBaggerState.eReady);
ELSE
	Ready := TRUE;	
END_IF
END_GET
END_PROPERTY

END_FUNCTION_BLOCK

// ---- POUs/GoodULStation_1.TcPOU
FUNCTION_BLOCK PUBLIC GoodULStation_1
VAR_INPUT
END_VAR
VAR_OUTPUT
END_VAR
VAR
	xTrigger :BOOL := FALSE; // triggers processing
	State : eGoodULNewStaState := eGoodULNewStaState.eUnknown;
	NextState : eGoodULNewStaState := eGoodULNewStaState.eUnknown;
	ErrorReturnState : eGoodULNewStaState := eGoodULNewStaState.eUnknown;
	bFirst : BOOL := TRUE;
	VUT : BYTE; //VehicleID Under Station
	DwellTimer : TON;
	StateTimer : TON;
END_VAR

IF (GVL_IO.MachineEStopped) THEN 
	State := eGoodULNewStaState.eUnknown;
	NextState := eGoodULNewStaState.eUnknown;
	Status.GoodUL_1_StatusMsg:= 'Good UL1 Sta Unknown, Check AIR, E-STOP and Hit Start';
END_IF

CASE State OF
eGoodULNewStaState.eUnknown:
	Status.GoodUL_1_StatusMsg:= 'Good UL1 Unknown, Check AIR, E-STOP and Hit Start';
    IF (GVL_IO.MC_XStartPB AND GVL_IO.MC_XAirPressureOK AND GVL_IO.MC_NotEStopped) THEN // wait for start button when powered up or PLC program restarted
		NextState := eGoodULNewStaState.eInit;	   
	END_IF
    

eGoodULNewStaState.eInit:
    Act_KnockPartOFF();
	Act_FreePalletHoldDown();
	ResetDwellTimer();
	NextState := eGoodULNewStaState.eHoming;
	

eGoodULNewStaState.eHoming:
	IF (IsPalletHoldDownFree()) THEN 
         NextState := eGoodULNewStaState.eReady;
	  END_IF
     DwellTimer(IN:=TRUE, PT:= T#10S);
     IF (DwellTimer.Q) THEN
		 ResetDwellTimer();
		 ErrorReturnState:= eGoodULNewStaState.eInit;
		 NextState := eGoodULNewStaState.eError;		 
	 END_IF	

eGoodULNewStaState.eReady:
	IF (xTrigger) THEN
		IF (NOT LotsData.Lot.AutoBaggerEnabled) THEN 
			Stations.fbRoutePlanner.P_GoodUnload_1_NextStaFlag := 5; 
			NextState := eGoodULNewStaState.eSendPalletHoldDownExtend;	
        ELSE
			NextState := eGoodULNewStaState.eCheckChuteCount;	
		END_IF		
		ResetDwellTimer();
	END_IF
	
	IF (NOT LotsData.Lot.GoodUnloadEnabled) THEN
		NextState :=  eGoodULNewStaState.eDisabledReady;	
	END_IF

eGoodULNewStaState.eDisabledReady:

	Act_KnockPartOFF();
	Act_FreePalletHoldDown();
	
    IF (LotsData.Lot.GoodUnloadEnabled) THEN 
		NextState := eGoodULNewStaState.eUnknown; // force the operator to hit the start button if station is enabled.
	END_IF
	
    IF (xTrigger) THEN // vehicles that have been previously commanded to come here before station was disabled 
		Stations.fbRoutePlanner.P_GoodUnload_1_NextStaFlag := 5; //// send to reject after this process is complete
		NextState := eGoodULNewStaState.eDepart;
	END_IF
	
	Status.StationStauts[MM_CONST.GOOD_UL_1_STA_HMI_STATE] := OverallStationStatus.eDisabled;
	Status.GoodUL_1_StatusMsg:= 'Good UL1 Disabled and Clear for pallets to move';	

eGoodULNewStaState.eCheckChuteCount: 
	IF ((Config.PremiumCount1 < LotsData.Lot.QuantityInBag) AND (Config.PremiumCount2 < (LotsData.Lot.QuantityInBag-10) OR Config.PremiumCount2 = LotsData.Lot.QuantityInBag )) THEN
			Stations.fbRoutePlanner.P_GoodUnload_1_NextStaFlag := 5; // send to reject after this process is complete
			NextState := eGoodULNewStaState.eSendPalletHoldDownExtend;	
            			
	ELSE 	
			Stations.fbRoutePlanner.P_GoodUnload_1_NextStaFlag := 2; // send to Good Unload Station 2
			NextState := eGoodULNewStaState.eDepart;
	END_IF

eGoodULNewStaState.eSendPalletHoldDownExtend:
	Act_EngagePalletHoldDown();
	ResetDwellTimer();
	NextState := eGoodULNewStaState.eCheckPalletHoldDownExtended;
	
eGoodULNewStaState.eCheckPalletHoldDownExtended:
   DwellTimer(IN:=TRUE, PT:= T#10S);	
   IF (IsPalletHoldDownEngaged()) THEN
        ResetDwellTimer();	   
		IF(GVL_IO.UL_1_XBarrelPresent (*OR TRUE*)) THEN    /// enabled checking Part Present Sensor at Unload stations 051319 NAP
			NextState := eGoodULNewStaState.eKnockOffPart;
        ELSE
			NextState := eGoodULNewStaState.ePalletHoldDownRelease;	
		END_IF        
   END_IF      
   IF (DwellTimer.Q) THEN
		 ResetDwellTimer();
		 ErrorReturnState:= eGoodULNewStaState.eSendPalletHoldDownExtend;
		 NextState := eGoodULNewStaState.eError;		 
	END_IF
  
eGoodULNewStaState.eKnockoffPart:
	Act_KnockPartON();
	UpdateLotData();
	UpdatePartData();
	ResetDwellTimer();
	StateTimer(IN:=FALSE);
	NextState := eGoodULNewStaState.eCheckPartKnockedOff;	

eGoodULNewStaState.eCheckPartKnockedOff:
   StateTimer(IN:=TRUE, PT:= T#200MS);
   IF (StateTimer.Q) THEN
   //IF (NOT(GVL_IO.UL_1_XBarrelPresent) ) THEN   
	   NextState := eGoodULNewStaState.ePalletHoldDownRelease;
	   Config.PremiumCount1 := Config.PremiumCount1 + 1;
	   DwellTimer(IN:=FALSE);
	   StateTimer(IN:=FALSE);
   END_IF
   DwellTimer(IN:= TRUE, PT:= T#10S);
   IF (DwellTimer.Q) THEN
	   ResetDwellTimer();
	   ErrorReturnState:= eGoodULNewStaState.eCheckPartKnockedOff;
	   Status.GoodUL_1_StatusMsg:= 'Good UL1 Remove Part then Hit START';
   	   NextState := eGoodULNewStaState.eError;	
   END_IF   

eGoodULNewStaState.ePalletHoldDownRelease:
    Act_KnockPartOFF();
	Act_FreePalletHoldDown();
    ResetDwellTimer();	
	NextState := eGoodULNewStaState.ePalletHoldDownReleased;

eGoodULNewStaState.ePalletHoldDownReleased:	
	IF (IsPalletHoldDownFree()) THEN         
	    NextState := eGoodULNewStaState.eDepart;
    END_IF
	
   DwellTimer(IN:= TRUE, PT:= T#10S);
   IF (DwellTimer.Q) THEN
	   ResetDwellTimer();
	   ErrorReturnState:= eGoodULNewStaState.ePalletHoldDownRelease;	   
   	   NextState := eGoodULNewStaState.eError;	
   END_IF  
	
	
eGoodULNewStaState.eDepart:
    Stations.fbRoutePlanner.M_NotifyVehStaCmpl(StationIndex:= MM_CONST.GOOD_UL_1_STA, VehicleID := VUT);
	xTrigger := FALSE;
	IF (Stations.fbCycleControl.StopRequested) THEN
		NextState := eGoodULNewStaState.eStopActive;
	ELSE 
		NextState := eGoodULNewStaState.eReady;
    END_IF
	
eGoodULNewStaState.eStopActive:
	IF (NOT Stations.fbCycleControl.StopRequested) THEN
		NextState := eGoodULNewStaState.eInit;
    END_IF
	

eGoodULNewStaState.eError:
	IF (GVL_IO.MC_XStartPB) THEN
		NextState := ErrorReturnState;
		ErrorReturnState := eGoodULNewStaState.eUnknown;
	END_IF

END_CASE

IF (State <> NextState) THEN
	bFirst := TRUE;
	StateTimer(IN:=FALSE);
ELSE
	bFirst := FALSE;
END_IF

State := NextState;
AssignStationStatusForHMI();

ACTION Act_EngagePalletHoldDown:
GVL_IO.UL_1_YPalletHoldDownExtend_Home  := FALSE;
GVL_IO.UL_1_YPalletHoldDownRetract_Engage := TRUE;
END_ACTION

ACTION Act_FreePalletHoldDown:
GVL_IO.UL_1_YPalletHoldDownExtend_Home := TRUE;
GVL_IO.UL_1_YPalletHoldDownRetract_Engage := FALSE;
END_ACTION

ACTION Act_KnockPartOFF:
GVL_IO.UL_1_YRejectPushExtend := FALSE;
GVL_IO.UL_1_YRejectPushRetract := TRUE;
END_ACTION

ACTION Act_KnockPartON:
GVL_IO.UL_1_YRejectPushExtend := TRUE;
GVL_IO.UL_1_YRejectPushRetract := FALSE;
END_ACTION

METHOD PUBLIC AssignStationStatusForHMI : BOOL
VAR_INPUT
END_VAR
Status.StationsState[MM_CONST.GOOD_UL_1_STA_HMI_STATE] := State;
IF (NOT LotsData.Lot.GoodUnloadEnabled) THEN
	Status.StationStauts[MM_CONST.GOOD_UL_1_STA_HMI_STATE] := OverallStationStatus.eDisabled;
ELSE 
	CASE State OF 
	
	eGoodULNewStaState.eUnknown,eGoodULNewStaState.eError:
		Status.StationStauts[MM_CONST.GOOD_UL_1_STA_HMI_STATE] := OverallStationStatus.eError;
		
    eGoodULNewStaState.eInit,
	eGoodULNewStaState.eHoming:
	    Status.StationStauts[MM_CONST.GOOD_UL_1_STA_HMI_STATE] := OverallStationStatus.eHoming;
	
	eGoodULNewStaState.eReady,eGoodULNewStaState.eWaitForVehicleTrigger:
	     Status.StationStauts[MM_CONST.GOOD_UL_1_STA_HMI_STATE] := OverallStationStatus.eWaitingForParts;
		 
	eGoodULNewStaState.eDwell,
	eGoodULNewStaState.eSendPalletHoldDownExtend,
	eGoodULNewStaState.eCheckPalletHoldDownExtended,
	eGoodULNewStaState.ePalletReleaseExtend,
	eGoodULNewStaState.ePalletReleaseExtended,
	eGoodULNewStaState.eKnockoffPart,
	eGoodULNewStaState.eKnockoffExtended,
	eGoodULNewStaState.eCheckPartKnockedOff,
	eGoodULNewStaState.ePalletHoldDownRelease,
	eGoodULNewStaState.ePalletHoldDownReleased:
	    Status.StationStauts[MM_CONST.GOOD_UL_1_STA_HMI_STATE] := OverallStationStatus.eRunning;
	
	eGoodULNewStaState.eStopActive:
	    Status.StationStauts[MM_CONST.GOOD_UL_1_STA_HMI_STATE] := OverallStationStatus.eCycleStop;
    	
	
    ELSE;	
	END_CASE
END_IF
END_METHOD

METHOD PUBLIC ClearVehicleTrigger : BOOL
VAR_INPUT
END_VAR
xTrigger := FALSE;
END_METHOD

METHOD PUBLIC IsFaulted : BOOL
VAR_INPUT
END_VAR
IsFaulted := (State = eGoodULNewStaState.eUnknown OR State = eGoodULNewStaState.eError);
END_METHOD

METHOD PUBLIC IsPalletHoldDownEngaged : BOOL
VAR_INPUT
END_VAR
IsPalletHoldDownEngaged := (GVL_IO.UL_1_XPalletHoldDownRetracted_Engaged AND NOT GVL_IO.UL_1_XPalletHoldDownExtended_Home);
IF (NOT IsPalletHoldDownEngaged) THEN
	Status.GoodUL_1_StatusMsg:= 'Good UL 1: Check Pallet Hold Down Sensors and then hit START';
END_IF
END_METHOD

METHOD PUBLIC IsPalletHoldDownFree : BOOL
VAR_INPUT
END_VAR
IsPalletHoldDownFree := (NOT GVL_IO.UL_1_XPalletHoldDownRetracted_Engaged AND GVL_IO.UL_1_XPalletHoldDownExtended_Home);
IF (NOT IsPalletHoldDownFree) THEN
	Status.GoodUL_1_StatusMsg := 'Good UL 1: Check Pallet Hold Down Sensors and then hit START';
END_IF
END_METHOD

PROPERTY PUBLIC Ready : BOOL
GET
IF (LotsData.Lot.GoodUnloadEnabled) THEN
	Ready := (State = eGoodULNewStaState.eReady);
ELSE
	Ready := (State = eGoodULNewStaState.eDisabledReady); 
END_IF
END_GET
END_PROPERTY

ACTION ResetDwellTimer:
DwellTimer(IN:=FALSE);
END_ACTION

METHOD PUBLIC ResetState : BOOL
VAR_INPUT
END_VAR
State := eGoodULNewStaState.eUnknown;
NextState := eGoodULNewStaState.eUnknown;
END_METHOD

PROPERTY PUBLIC Trigger : BOOL
SET
xTrigger := Trigger;
END_SET
END_PROPERTY

METHOD PUBLIC UpdateLotData : BOOL
VAR_INPUT
END_VAR
IF (PartsData.Status[VUT].Premium) THEN
	LotsData.Lot.CavityCounts[PartsData.Status[VUT].CavityNumber].PremiumCount := LotsData.Lot.CavityCounts[PartsData.Status[VUT].CavityNumber].PremiumCount +1;
ELSIF (PartsData.Status[VUT].Good) THEN
 	LotsData.Lot.CavityCounts[PartsData.Status[VUT].CavityNumber].GoodCount := LotsData.Lot.CavityCounts[PartsData.Status[VUT].CavityNumber].GoodCount + 1;
END_IF
LotsData.Lot.CavityCounts[PartsData.Status[VUT].CavityNumber].TotalCount := LotsData.Lot.CavityCounts[PartsData.Status[VUT].CavityNumber].TotalCount + 1;
 // reject parts shouldn't get here. If this station rejects something (e.g. faults out) then it barrel will go to reject station.
END_METHOD

METHOD PUBLIC UpdatePartData : BOOL
VAR_INPUT
END_VAR
PartsData.Status[VUT].UnloadTime := SYSTEMTIME_TO_STRING(Logging.fbCurrTime.systemTime);
PartsData.Status[VUT].OverallStatus := ePartStatus.eEmpty;
PartsData.Status[VUT].GoodUnload := TRUE;

// we will write data to CSV file over here 
IF (P_TextModeWrite.CurrWriteStep = 0) THEN 
	P_TextModeWrite.VehicleID := VUT;
	P_TextModeWrite.WriteData := TRUE;
END_IF
END_METHOD

PROPERTY PUBLIC VehicleUnderTest : BYTE
GET
VehicleUnderTest := VUT;
END_GET
SET
VUT := VehicleUnderTest;
END_SET
END_PROPERTY

END_FUNCTION_BLOCK

// ---- POUs/GoodULStation_2.TcPOU
FUNCTION_BLOCK PUBLIC GoodULStation_2
VAR_INPUT
END_VAR
VAR_OUTPUT
END_VAR
VAR
	xTrigger :BOOL := FALSE; // triggers processing
	State : eGoodULNewStaState := eGoodULNewStaState.eUnknown;
	NextState : eGoodULNewStaState := eGoodULNewStaState.eUnknown;
	ErrorReturnState : eGoodULNewStaState := eGoodULNewStaState.eUnknown;
	bFirst : BOOL := TRUE;
	VUT : BYTE; //VehicleID Under Station
	DwellTimer : TON;
	StateTimer : TON;
END_VAR

IF (GVL_IO.MachineEStopped) THEN 
	State := eGoodULNewStaState.eUnknown;
	NextState := eGoodULNewStaState.eUnknown;
	Status.GoodUL_2_StatusMsg:= 'Good UL2 Sta Unknown, Check AIR, E-STOP and Hit Start';
END_IF

CASE State OF
eGoodULNewStaState.eUnknown:
	Status.GoodUL_2_StatusMsg:= 'Good UL2 Unknown, Check AIR, E-STOP and Hit Start';
    IF (GVL_IO.MC_XStartPB AND GVL_IO.MC_XAirPressureOK AND GVL_IO.MC_NotEStopped) THEN // wait for start button when powered up or PLC program restarted
		NextState := eGoodULNewStaState.eInit;	   
	END_IF
    

eGoodULNewStaState.eInit:
    Act_KnockPartOFF();
	Act_FreePalletHoldDown();
	ResetDwellTimer();
	NextState := eGoodULNewStaState.eHoming;
	

eGoodULNewStaState.eHoming:
	IF (IsPalletHoldDownFree()) THEN 
         NextState := eGoodULNewStaState.eReady;
	  END_IF
     DwellTimer(IN:=TRUE, PT:= T#10S);
     IF (DwellTimer.Q) THEN
		 ResetDwellTimer();
		 ErrorReturnState:= eGoodULNewStaState.eInit;
		 NextState := eGoodULNewStaState.eError;		 
	 END_IF	

eGoodULNewStaState.eReady:
	IF (xTrigger) THEN
		IF (NOT LotsData.Lot.AutoBaggerEnabled) THEN 
				Stations.fbRoutePlanner.P_GoodUnload_2_NextStaFlag := 5; 
				NextState := eGoodULNewStaState.eSendPalletHoldDownExtend;	
		ELSE
				NextState := eGoodULNewStaState.eCheckChuteCount;	
		END_IF	
		ResetDwellTimer();
	END_IF
	
	IF (NOT LotsData.Lot.GoodUnloadEnabled) THEN
		NextState :=  eGoodULNewStaState.eDisabledReady;	
	END_IF

eGoodULNewStaState.eDisabledReady:

	Act_KnockPartOFF();
	Act_FreePalletHoldDown();
	
    IF (LotsData.Lot.GoodUnloadEnabled) THEN 
		NextState := eGoodULNewStaState.eUnknown; // force the operator to hit the start button if station is enabled.
	END_IF
	
    IF (xTrigger) THEN // vehicles that have been previously commanded to come here before station was disabled 
	Stations.fbRoutePlanner.P_GoodUnload_2_NextStaFlag := 5; //// send to reject after this process is complete	
	NextState := eGoodULNewStaState.eDepart;
	END_IF
	
	Status.StationStauts[MM_CONST.GOOD_UL_2_STA_HMI_STATE] := OverallStationStatus.eDisabled;
	Status.GoodUL_2_StatusMsg:= 'Good UL2 Disabled and Clear for pallets to move';	

eGoodULNewStaState.eCheckChuteCount:
	IF  (Config.PremiumCount2 < LotsData.Lot.QuantityInBag)  THEN
			Stations.fbRoutePlanner.P_GoodUnload_2_NextStaFlag := 5; // send to reject after this process is complete
			NextState := eGoodULNewStaState.eSendPalletHoldDownExtend;	
            			
	ELSE 	
			Stations.fbRoutePlanner.P_GoodUnload_2_NextStaFlag := 3; // send to Good Unload Station 2
			PartsData.Status[VUT].OverallStatus := ePartStatus.eGoodRegular;
        	PartsData.Status[VUT].Good := TRUE;	
			PartsData.Status[VUT].Premium := FALSE;
			PartsData.Status[VUT].VisionPass := TRUE;			
			NextState := eGoodULNewStaState.eDepart;
	END_IF

eGoodULNewStaState.eSendPalletHoldDownExtend:
	Act_EngagePalletHoldDown();
	ResetDwellTimer();
	NextState := eGoodULNewStaState.eCheckPalletHoldDownExtended;
	
eGoodULNewStaState.eCheckPalletHoldDownExtended:
   DwellTimer(IN:=TRUE, PT:= T#10S);	
   IF (IsPalletHoldDownEngaged()) THEN
        ResetDwellTimer();	   
		IF(GVL_IO.UL_2_XBarrelPresent (* OR TRUE*) ) THEN   /// enabled checking Part Present Sensor at Unload stations 051319 NAP
			NextState := eGoodULNewStaState.eKnockOffPart;
        ELSE
			NextState := eGoodULNewStaState.ePalletHoldDownRelease;	
		END_IF        
   END_IF      
   IF (DwellTimer.Q) THEN
		 ResetDwellTimer();
		 ErrorReturnState:= eGoodULNewStaState.eSendPalletHoldDownExtend;
		 NextState := eGoodULNewStaState.eError;		 
	END_IF
  
eGoodULNewStaState.eKnockoffPart:
	Act_KnockPartON();
	UpdateLotData();
	UpdatePartData();
	ResetDwellTimer();
	StateTimer(IN:=FALSE);
	NextState := eGoodULNewStaState.eCheckPartKnockedOff;

eGoodULNewStaState.eCheckPartKnockedOff:
	StateTimer(IN:=TRUE, PT:= T#200MS);
   	IF (StateTimer.Q) THEN
   //IF (NOT(GVL_IO.UL_2_XBarrelPresent) ) THEN   
	   NextState := eGoodULNewStaState.ePalletHoldDownRelease;
	   Config.PremiumCount2 := Config.PremiumCount2 + 1;
	   DwellTimer(IN:=FALSE);
	   StateTimer(IN:=FALSE);
   END_IF
   DwellTimer(IN:= TRUE, PT:= T#10S);
   IF (DwellTimer.Q) THEN
	   ResetDwellTimer();
	   ErrorReturnState:= eGoodULNewStaState.eCheckPartKnockedOff;
	   Status.GoodUL_2_StatusMsg:= 'Good UL 2 Remove Part then Hit START';
   	   NextState := eGoodULNewStaState.eError;	
   END_IF   

eGoodULNewStaState.ePalletHoldDownRelease:
    Act_KnockPartOFF();
	Act_FreePalletHoldDown();
    ResetDwellTimer();	
	NextState := eGoodULNewStaState.ePalletHoldDownReleased;

eGoodULNewStaState.ePalletHoldDownReleased:	
	IF (IsPalletHoldDownFree()) THEN         
	    NextState := eGoodULNewStaState.eDepart;
    END_IF
	
   DwellTimer(IN:= TRUE, PT:= T#10S);
   IF (DwellTimer.Q) THEN
	   ResetDwellTimer();
	   ErrorReturnState:= eGoodULNewStaState.ePalletHoldDownRelease;	   
   	   NextState := eGoodULNewStaState.eError;	
   END_IF  
	
	
eGoodULNewStaState.eDepart:
    Stations.fbRoutePlanner.M_NotifyVehStaCmpl(StationIndex:= MM_CONST.GOOD_UL_2_STA, VehicleID := VUT);
	xTrigger := FALSE;
	IF (Stations.fbCycleControl.StopRequested) THEN
		NextState := eGoodULNewStaState.eStopActive;
	ELSE 
		NextState := eGoodULNewStaState.eReady;
    END_IF
	
eGoodULNewStaState.eStopActive:
	IF (NOT Stations.fbCycleControl.StopRequested) THEN
		NextState := eGoodULNewStaState.eInit;
    END_IF
	

eGoodULNewStaState.eError:
	IF (GVL_IO.MC_XStartPB) THEN
		NextState := ErrorReturnState;
		ErrorReturnState := eGoodULNewStaState.eUnknown;
	END_IF

END_CASE

IF (State <> NextState) THEN
	bFirst := TRUE;
	StateTimer(IN:=FALSE);
ELSE
	bFirst := FALSE;
END_IF

State := NextState;
AssignStationStatusForHMI();

ACTION Act_EngagePalletHoldDown:
GVL_IO.UL_2_YPalletHoldDownExtend_Home  := FALSE;
GVL_IO.UL_2_YPalletHoldDownRetract_Engage := TRUE;
END_ACTION

ACTION Act_FreePalletHoldDown:
GVL_IO.UL_2_YPalletHoldDownExtend_Home := TRUE;
GVL_IO.UL_2_YPalletHoldDownRetract_Engage := FALSE;
END_ACTION

ACTION Act_KnockPartOFF:
GVL_IO.UL_2_YRejectPushExtend := FALSE;
GVL_IO.UL_2_YRejectPushRetract := TRUE;
END_ACTION

ACTION Act_KnockPartON:
GVL_IO.UL_2_YRejectPushExtend := TRUE;
GVL_IO.UL_2_YRejectPushRetract := FALSE;
END_ACTION

METHOD PUBLIC AssignStationStatusForHMI : BOOL
VAR_INPUT
END_VAR
Status.StationsState[MM_CONST.GOOD_UL_2_STA_HMI_STATE] := State;
IF (NOT LotsData.Lot.GoodUnloadEnabled) THEN
	Status.StationStauts[MM_CONST.GOOD_UL_2_STA_HMI_STATE] := OverallStationStatus.eDisabled;
ELSE 
	CASE State OF 
	
	eGoodULNewStaState.eUnknown,eGoodULNewStaState.eError:
		Status.StationStauts[MM_CONST.GOOD_UL_2_STA_HMI_STATE] := OverallStationStatus.eError;
		
    eGoodULNewStaState.eInit,
	eGoodULNewStaState.eHoming:
	    Status.StationStauts[MM_CONST.GOOD_UL_2_STA_HMI_STATE] := OverallStationStatus.eHoming;
	
	eGoodULNewStaState.eReady,eGoodULNewStaState.eWaitForVehicleTrigger:
	     Status.StationStauts[MM_CONST.GOOD_UL_2_STA_HMI_STATE] := OverallStationStatus.eWaitingForParts;
		 
	eGoodULNewStaState.eDwell,
	eGoodULNewStaState.eSendPalletHoldDownExtend,
	eGoodULNewStaState.eCheckPalletHoldDownExtended,
	eGoodULNewStaState.ePalletReleaseExtend,
	eGoodULNewStaState.ePalletReleaseExtended,
	eGoodULNewStaState.eKnockoffPart,
	eGoodULNewStaState.eKnockoffExtended,
	eGoodULNewStaState.eCheckPartKnockedOff,
	eGoodULNewStaState.ePalletHoldDownRelease,
	eGoodULNewStaState.ePalletHoldDownReleased:
	    Status.StationStauts[MM_CONST.GOOD_UL_2_STA_HMI_STATE] := OverallStationStatus.eRunning;
	
	eGoodULNewStaState.eStopActive:
	    Status.StationStauts[MM_CONST.GOOD_UL_2_STA_HMI_STATE] := OverallStationStatus.eCycleStop;
    	
	
    ELSE;	
	END_CASE
END_IF
END_METHOD

METHOD PUBLIC ClearVehicleTrigger : BOOL
VAR_INPUT
END_VAR
xTrigger := FALSE;
END_METHOD

METHOD PUBLIC IsFaulted : BOOL
VAR_INPUT
END_VAR
IsFaulted := (State = eGoodULNewStaState.eUnknown OR State = eGoodULNewStaState.eError);
END_METHOD

METHOD PUBLIC IsPalletHoldDownEngaged : BOOL
VAR_INPUT
END_VAR
IsPalletHoldDownEngaged := (GVL_IO.UL_2_XPalletHoldDownRetracted_Engaged AND NOT GVL_IO.UL_2_XPalletHoldDownExtended_Home);
IF (NOT IsPalletHoldDownEngaged) THEN
	Status.GoodUL_2_StatusMsg:= 'Good UL 2: Check Pallet Hold Down Sensors and then hit START';
END_IF
END_METHOD

METHOD PUBLIC IsPalletHoldDownFree : BOOL
VAR_INPUT
END_VAR
IsPalletHoldDownFree := (NOT GVL_IO.UL_2_XPalletHoldDownRetracted_Engaged AND GVL_IO.UL_2_XPalletHoldDownExtended_Home);
IF (NOT IsPalletHoldDownFree) THEN
	Status.GoodUL_2_StatusMsg := 'Good UL 2: Check Pallet Hold Down Sensors and then hit START';
END_IF
END_METHOD

PROPERTY PUBLIC Ready : BOOL
GET
IF (LotsData.Lot.GoodUnloadEnabled) THEN
	Ready := (State = eGoodULNewStaState.eReady);
ELSE
	Ready := (State = eGoodULNewStaState.eDisabledReady); 
END_IF
END_GET
END_PROPERTY

ACTION ResetDwellTimer:
DwellTimer(IN:=FALSE);
END_ACTION

METHOD PUBLIC ResetState : BOOL
VAR_INPUT
END_VAR
State := eGoodULNewStaState.eUnknown;
NextState := eGoodULNewStaState.eUnknown;
END_METHOD

PROPERTY PUBLIC Trigger : BOOL
SET
xTrigger := Trigger;
END_SET
END_PROPERTY

METHOD PUBLIC UpdateLotData : BOOL
VAR_INPUT
END_VAR
IF (PartsData.Status[VUT].Premium) THEN
	LotsData.Lot.CavityCounts[PartsData.Status[VUT].CavityNumber].PremiumCount := LotsData.Lot.CavityCounts[PartsData.Status[VUT].CavityNumber].PremiumCount +1;
ELSIF (PartsData.Status[VUT].Good) THEN
 	LotsData.Lot.CavityCounts[PartsData.Status[VUT].CavityNumber].GoodCount := LotsData.Lot.CavityCounts[PartsData.Status[VUT].CavityNumber].GoodCount + 1;
END_IF
LotsData.Lot.CavityCounts[PartsData.Status[VUT].CavityNumber].TotalCount := LotsData.Lot.CavityCounts[PartsData.Status[VUT].CavityNumber].TotalCount + 1;
 // reject parts shouldn't get here. If this station rejects something (e.g. faults out) then it barrel will go to reject station.
END_METHOD

METHOD PUBLIC UpdatePartData : BOOL
VAR_INPUT
END_VAR
PartsData.Status[VUT].UnloadTime := SYSTEMTIME_TO_STRING(Logging.fbCurrTime.systemTime);
PartsData.Status[VUT].OverallStatus := ePartStatus.eEmpty;
PartsData.Status[VUT].GoodUnload := TRUE;

// we will write data to CSV file over here 
IF (P_TextModeWrite.CurrWriteStep = 0) THEN 
	P_TextModeWrite.VehicleID := VUT;
	P_TextModeWrite.WriteData := TRUE;
END_IF
END_METHOD

PROPERTY PUBLIC VehicleUnderTest : BYTE
GET
VehicleUnderTest := VUT;
END_GET
SET
VUT := VehicleUnderTest;
END_SET
END_PROPERTY

END_FUNCTION_BLOCK

// ---- POUs/GoodULStation_3.TcPOU
FUNCTION_BLOCK PUBLIC GoodULStation_3
VAR_INPUT
END_VAR
VAR_OUTPUT
END_VAR
VAR
	xTrigger :BOOL := FALSE; // triggers processing
	State : eGoodULNewStaState := eGoodULNewStaState.eUnknown;
	NextState : eGoodULNewStaState := eGoodULNewStaState.eUnknown;
	ErrorReturnState : eGoodULNewStaState := eGoodULNewStaState.eUnknown;
	bFirst : BOOL := TRUE;
	VUT : BYTE; //VehicleID Under Station
	DwellTimer : TON;
	StateTimer : TON;
END_VAR

IF (GVL_IO.MachineEStopped) THEN 
	State := eGoodULNewStaState.eUnknown;
	NextState := eGoodULNewStaState.eUnknown;
	Status.GoodUL_3_StatusMsg:= 'Good UL3 Sta Unknown, Check AIR, E-STOP and Hit Start';
END_IF

CASE State OF
eGoodULNewStaState.eUnknown:
	Status.GoodUL_3_StatusMsg:= 'Good UL3 Unknown, Check AIR, E-STOP and Hit Start';
    IF (GVL_IO.MC_XStartPB AND GVL_IO.MC_XAirPressureOK AND GVL_IO.MC_NotEStopped) THEN // wait for start button when powered up or PLC program restarted
		NextState := eGoodULNewStaState.eInit;	   
	END_IF
    

eGoodULNewStaState.eInit:
    Act_KnockPartOFF();
	Act_FreePalletHoldDown();
	ResetDwellTimer();
	NextState := eGoodULNewStaState.eHoming;
	

eGoodULNewStaState.eHoming:
	IF (IsPalletHoldDownFree()) THEN 
         NextState := eGoodULNewStaState.eReady;
	  END_IF
     DwellTimer(IN:=TRUE, PT:= T#10S);
     IF (DwellTimer.Q) THEN
		 ResetDwellTimer();
		 ErrorReturnState:= eGoodULNewStaState.eInit;
		 NextState := eGoodULNewStaState.eError;		 
	 END_IF	

eGoodULNewStaState.eReady:
	IF (xTrigger) THEN
		IF (NOT LotsData.Lot.AutoBaggerEnabled) THEN 
				Stations.fbRoutePlanner.P_GoodUnload_3_NextStaFlag := 5; 
				NextState := eGoodULNewStaState.eSendPalletHoldDownExtend;	
		ELSE
				NextState := eGoodULNewStaState.eCheckChuteCount;	
		END_IF	
		ResetDwellTimer();
	END_IF
	
	IF (NOT LotsData.Lot.GoodUnloadEnabled) THEN
		NextState :=  eGoodULNewStaState.eDisabledReady;	
	END_IF

eGoodULNewStaState.eDisabledReady:

	Act_KnockPartOFF();
	Act_FreePalletHoldDown();
	
    IF (LotsData.Lot.GoodUnloadEnabled) THEN 
		NextState := eGoodULNewStaState.eUnknown; // force the operator to hit the start button if station is enabled.
	END_IF
	
    IF (xTrigger) THEN // vehicles that have been previously commanded to come here before station was disabled 
		Stations.fbRoutePlanner.P_GoodUnload_3_NextStaFlag := 5; // send to reject after this process is complete
		NextState := eGoodULNewStaState.eDepart;
	END_IF
	
	Status.StationStauts[MM_CONST.GOOD_UL_3_STA_HMI_STATE] := OverallStationStatus.eDisabled;
	Status.GoodUL_3_StatusMsg:= 'Good UL3 Disabled and Clear for pallets to move';	

eGoodULNewStaState.eCheckChuteCount: 
	IF ((Config.GoodCount1 < LotsData.Lot.QuantityInBag) AND (Config.GoodCount2 < (LotsData.Lot.QuantityInBag-10) OR Config.GoodCount2 = LotsData.Lot.QuantityInBag)) THEN
			Stations.fbRoutePlanner.P_GoodUnload_3_NextStaFlag := 5; // send to reject after this process is complete
			NextState := eGoodULNewStaState.eSendPalletHoldDownExtend;	
            			
	ELSE 	
			Stations.fbRoutePlanner.P_GoodUnload_3_NextStaFlag := 4; // send to Good Unload Station 4
			NextState := eGoodULNewStaState.eDepart;
	END_IF
	
eGoodULNewStaState.eSendPalletHoldDownExtend:
	Act_EngagePalletHoldDown();
	ResetDwellTimer();
	NextState := eGoodULNewStaState.eCheckPalletHoldDownExtended;
	
eGoodULNewStaState.eCheckPalletHoldDownExtended:
   DwellTimer(IN:=TRUE, PT:= T#10S);	
   IF (IsPalletHoldDownEngaged()) THEN
        ResetDwellTimer();	   
		IF(GVL_IO.UL_3_XBarrelPresent (*OR TRUE*)) THEN   /// enabled checking Part Present Sensor at Unload stations 051319 NAP
			NextState := eGoodULNewStaState.eKnockOffPart;
        ELSE
			NextState := eGoodULNewStaState.ePalletHoldDownRelease;	
		END_IF        
   END_IF      
   IF (DwellTimer.Q) THEN
		 ResetDwellTimer();
		 ErrorReturnState:= eGoodULNewStaState.eSendPalletHoldDownExtend;
		 NextState := eGoodULNewStaState.eError;		 
	END_IF
  
eGoodULNewStaState.eKnockoffPart:
	Act_KnockPartON();
	UpdateLotData();
	UpdatePartData();
	ResetDwellTimer();
	StateTimer(IN:=FALSE);
	NextState := eGoodULNewStaState.eCheckPartKnockedOff;

eGoodULNewStaState.eCheckPartKnockedOff:
   StateTimer(IN:=TRUE, PT:= T#200MS);
   	IF (StateTimer.Q) THEN
   //IF (NOT(GVL_IO.UL_3_XBarrelPresent) ) THEN   
	   NextState := eGoodULNewStaState.ePalletHoldDownRelease;
	   Config.GoodCount1 := Config.GoodCount1 + 1;
	   DwellTimer(IN:=FALSE);
	   StateTimer(IN:=FALSE);
   END_IF
   DwellTimer(IN:= TRUE, PT:= T#10S);
   IF (DwellTimer.Q) THEN
	   ResetDwellTimer();
	   ErrorReturnState:= eGoodULNewStaState.eCheckPartKnockedOff;
	   Status.GoodUL_3_StatusMsg:= 'Good UL 3 Remove Part then Hit START';
   	   NextState := eGoodULNewStaState.eError;	
   END_IF   

eGoodULNewStaState.ePalletHoldDownRelease:
    Act_KnockPartOFF();
	Act_FreePalletHoldDown();
    ResetDwellTimer();	
	NextState := eGoodULNewStaState.ePalletHoldDownReleased;

eGoodULNewStaState.ePalletHoldDownReleased:	
	IF (IsPalletHoldDownFree()) THEN         
	    NextState := eGoodULNewStaState.eDepart;
    END_IF
	
   DwellTimer(IN:= TRUE, PT:= T#10S);
   IF (DwellTimer.Q) THEN
	   ResetDwellTimer();
	   ErrorReturnState:= eGoodULNewStaState.ePalletHoldDownRelease;	   
   	   NextState := eGoodULNewStaState.eError;	
   END_IF  
	
	
eGoodULNewStaState.eDepart:
    Stations.fbRoutePlanner.M_NotifyVehStaCmpl(StationIndex:= MM_CONST.GOOD_UL_3_STA, VehicleID := VUT);
	xTrigger := FALSE;
	IF (Stations.fbCycleControl.StopRequested) THEN
		NextState := eGoodULNewStaState.eStopActive;
	ELSE 
		NextState := eGoodULNewStaState.eReady;
    END_IF
	
eGoodULNewStaState.eStopActive:
	IF (NOT Stations.fbCycleControl.StopRequested) THEN
		NextState := eGoodULNewStaState.eInit;
    END_IF
	

eGoodULNewStaState.eError:
	IF (GVL_IO.MC_XStartPB) THEN
		NextState := ErrorReturnState;
		ErrorReturnState := eGoodULNewStaState.eUnknown;
	END_IF

END_CASE

IF (State <> NextState) THEN
	bFirst := TRUE;
	StateTimer(IN:=FALSE);
ELSE
	bFirst := FALSE;
END_IF

State := NextState;
AssignStationStatusForHMI();

ACTION Act_EngagePalletHoldDown:
GVL_IO.UL_3_YPalletHoldDownExtend_Home  := FALSE;
GVL_IO.UL_3_YPalletHoldDownRetract_Engage := TRUE;
END_ACTION

ACTION Act_FreePalletHoldDown:
GVL_IO.UL_3_YPalletHoldDownExtend_Home := TRUE;
GVL_IO.UL_3_YPalletHoldDownRetract_Engage := FALSE;
END_ACTION

ACTION Act_KnockPartOFF:
GVL_IO.UL_3_YRejectPushExtend := FALSE;
GVL_IO.UL_3_YRejectPushRetract := TRUE;
END_ACTION

ACTION Act_KnockPartON:
GVL_IO.UL_3_YRejectPushExtend := TRUE;
GVL_IO.UL_3_YRejectPushRetract := FALSE;
END_ACTION

METHOD PUBLIC AssignStationStatusForHMI : BOOL
VAR_INPUT
END_VAR
Status.StationsState[MM_CONST.GOOD_UL_3_STA_HMI_STATE] := State;
IF (NOT LotsData.Lot.GoodUnloadEnabled) THEN
	Status.StationStauts[MM_CONST.GOOD_UL_3_STA_HMI_STATE] := OverallStationStatus.eDisabled;
ELSE 
	CASE State OF 
	
	eGoodULNewStaState.eUnknown,eGoodULNewStaState.eError:
		Status.StationStauts[MM_CONST.GOOD_UL_3_STA_HMI_STATE] := OverallStationStatus.eError;
		
    eGoodULNewStaState.eInit,
	eGoodULNewStaState.eHoming:
	    Status.StationStauts[MM_CONST.GOOD_UL_3_STA_HMI_STATE] := OverallStationStatus.eHoming;
	
	eGoodULNewStaState.eReady,eGoodULNewStaState.eWaitForVehicleTrigger:
	     Status.StationStauts[MM_CONST.GOOD_UL_3_STA_HMI_STATE] := OverallStationStatus.eWaitingForParts;
		 
	eGoodULNewStaState.eDwell,
	eGoodULNewStaState.eSendPalletHoldDownExtend,
	eGoodULNewStaState.eCheckPalletHoldDownExtended,
	eGoodULNewStaState.ePalletReleaseExtend,
	eGoodULNewStaState.ePalletReleaseExtended,
	eGoodULNewStaState.eKnockoffPart,
	eGoodULNewStaState.eKnockoffExtended,
	eGoodULNewStaState.eCheckPartKnockedOff,
	eGoodULNewStaState.ePalletHoldDownRelease,
	eGoodULNewStaState.ePalletHoldDownReleased:
	    Status.StationStauts[MM_CONST.GOOD_UL_3_STA_HMI_STATE] := OverallStationStatus.eRunning;
	
	eGoodULNewStaState.eStopActive:
	    Status.StationStauts[MM_CONST.GOOD_UL_3_STA_HMI_STATE] := OverallStationStatus.eCycleStop;
    	
	
    ELSE;	
	END_CASE
END_IF
END_METHOD

METHOD PUBLIC ClearVehicleTrigger : BOOL
VAR_INPUT
END_VAR
xTrigger := FALSE;
END_METHOD

